# B&R Automation Studio project RS15_RX_30005_r00 (part 7)

#### Control.var
```iecst
(********************************************************************
 * COPYRIGHT -- .
 ********************************************************************
 * Program: Control
 * File: Control.var
 * Author: dominique
 * Created: August 16, 2011
 ********************************************************************
 * Local variables of program Control
 ********************************************************************)

VAR
  bHMI_Bund_ManOn_PB : BOOL ; (*Bundler lacal manuel mode, =0:Off; =1:On*)
  bHMI_Bund_Init_PB  : BOOL ;
  bBundManOn         : BOOL ;
  bBundManOff        : BOOL ;
  bInitBund          : BOOL ;
  bInitBundStart     : BOOL ;
  bInitBundStop      : BOOL ;
  uiBundManTxt_Ind   : UINT ;
  uiBundManCol_Ind   : UINT ;
  uiBundInitTxt_Ind  : UINT ;
  uiBundInitCol_Ind  : UINT ;
  tBundInitTpHorn    : TIME ;

  bHMI_Bund_OnOff  : BOOL ;
  iHMI_BundManLock : INT ;

  H_FB_ToggleTB_0 : H_FB_ToggleTB;

  bBundInit_Perm   : BOOL ;
  H_FB_2StepMove_0 : H_FB_2StepMove ;

  stTP_0 : TP ;
END_VAR

VAR CONSTANT

END_VAR
```

#### ControlInit.st
```iecst
(********************************************************************
 * COPYRIGHT -- .
 ********************************************************************
 * Program: Control
 * File: ControlInit.st
 * Author: dominique
 * Created: August 16, 2011
 ********************************************************************
 * Implementation of program Control
 ********************************************************************)

PROGRAM _INIT

// Bundler Manual/Auto TB Colors
  H_FB_ToggleTB_0.IN_uiTxt0_Ind := 0 ;
  H_FB_ToggleTB_0.IN_uiTxt1_Ind := -1 ;
  H_FB_ToggleTB_0.IN_uiBackCol_State0 := gYellow;
  H_FB_ToggleTB_0.IN_uiForeCol_State0 := gBlack;
  H_FB_ToggleTB_0.IN_uiBackCol_State1 := gGreen;
  H_FB_ToggleTB_0.IN_uiForeCol_State1 := gBlack;

  tBundInitTpHorn     := T#1s ;
  g_tBund_TpWatchSens := T#3s ;

  bHMI_Bund_OnOff := 0 ;

END_PROGRAM
```

### Program Logical/BagMachine_Section/BagBundler/Separator (IEC)

#### SeparatorCyclic.st - Cyclic code
```iecst
(********************************************************************
 * COPYRIGHT -- .
 ********************************************************************
 * Program: Separator
 * File: SeparatorCyclic.st
 * Author: dominique
 * Created: August 15, 2011
 ********************************************************************
 * Implementation of program Separator
 ********************************************************************)

PROGRAM _CYCLIC

    //---------------------------------------------------------------------------------------------------------------------
    // Output assignments
    gQ_Bund_SOL_14C1Out    := bQ_Bund_SOL_14C1Out AND gBagMachine_EstopAlarmsOK ;
    gQ_Bund_SOL_14C2Out    := bQ_Bund_SOL_14C2Out AND gBagMachine_EstopAlarmsOK ;
    gQ_Bund_SOL_PresSelect := bQ_Bund_SOL_PresSelect AND gBagMachine_EstopAlarmsOK ;

    //---------------------------------------------------------------------------------------------------------------------
    // Sensor watching

    H_FB_Flash_0(IN_bEnable:=1, IN_rNumFlashPerSec:=2) ;
    bFlash := H_FB_Flash_0.OUT_bFlash ;

    // S102 on 14C1 Out
    H_FB_WS_14C1.IN_bSensorOut  := gI_Bund_S102 ;
    H_FB_WS_14C1.IN_bSOL_In     := NOT(gQ_Bund_SOL_14C1Out) ;
    H_FB_WS_14C1.IN_bSOL_Out    := gQ_Bund_SOL_14C1Out ;
    H_FB_WS_14C1.IN_bActSensIn  := 0 ;
    H_FB_WS_14C1.IN_bActSensOut := 1 ;
    H_FB_WS_14C1.IN_tTpWatchIn  := g_tBund_TpWatchSens ;
    H_FB_WS_14C1.IN_tTpWatchOut := g_tBund_TpWatchSens ;
    H_FB_WS_14C1.IN_bReset      := gAlarmReset ;
    H_FB_WS_14C1();
    bS102_FaultOut := H_FB_WS_14C1.OUT_bSensOut_FaultOut ;
    bS102_FaultIn  := H_FB_WS_14C1.OUT_bSensOut_FaultIn ;
    bS102_Fault    := H_FB_WS_14C1.OUT_bSensOut_Fault ;

    // S101 on 14C2 In
    H_FB_WS_14C2.IN_bSensorIn   := gI_Bund_S101 ;
    H_FB_WS_14C2.IN_bSOL_In     := NOT(gQ_Bund_SOL_14C2Out) ;
    H_FB_WS_14C2.IN_bSOL_Out    := gQ_Bund_SOL_14C2Out ;
    H_FB_WS_14C2.IN_bActSensIn  := 1 ;
    H_FB_WS_14C2.IN_bActSensOut := 0 ;
    H_FB_WS_14C2.IN_tTpWatchIn  := g_tBund_TpWatchSens ;
    H_FB_WS_14C2.IN_tTpWatchOut := g_tBund_TpWatchSens ;
    H_FB_WS_14C2.IN_bReset      := gAlarmReset ;
    H_FB_WS_14C2();
    bS101_FaultOut := H_FB_WS_14C2.OUT_bSensIn_FaultOut ;
    bS101_FaultIn  := H_FB_WS_14C2.OUT_bSensIn_FaultIn ;
    bS101_Fault    := H_FB_WS_14C2.OUT_bSensIn_Fault ;

    // HMI Sensors states display
    IF gI_Bund_S101 THEN
      iHMI_Bund_S101 := 1 ;
    ELSE
      iHMI_Bund_S101 := 0 ;
    END_IF
    IF bS101_Fault AND
       bFlash      THEN
      iHMI_Bund_S101 := 2 ;
    END_IF

    IF gI_Bund_S102 THEN
      iHMI_Bund_S102 := 1 ;
    ELSE
      iHMI_Bund_S102 := 0 ;
    END_IF
    IF bS102_Fault AND
       bFlash      THEN
      iHMI_Bund_S102 := 2 ;
    END_IF

    IF gI_Bund_S103 THEN
      iHMI_Bund_S103 := 1 ;
    ELSE
      iHMI_Bund_S103 := 0 ;
    END_IF

    IF gI_Bund_S109 THEN
      iHMI_Bund_S109 := 1 ;
    ELSE
      iHMI_Bund_S109 := 0 ;
    END_IF

    g_bBund_SensFaultCycSep := bS101_Fault OR bS102_Fault ;

    // HMI Cylinders states display
    // Cylinder 14C1
    // Case Out
    IF gQ_Bund_SOL_14C1Out THEN
      iHMI_Bund_14C1Out_State := 4 ;
      iHMI_Bund_14C1In_State  := 0 ;
    END_IF
    IF bS102_FaultOut THEN
      IF bFlash THEN
        iHMI_Bund_14C1Out_State := 5 ;
      ELSE
        iHMI_Bund_14C1Out_State := 6 ;
      END_IF
    END_IF
    // Case In
    IF NOT(gQ_Bund_SOL_14C1Out) THEN
      iHMI_Bund_14C1In_State  := 1 ;
      iHMI_Bund_14C1Out_State := 0 ;
    END_IF
    IF bS102_FaultIn THEN
      IF bFlash THEN
        iHMI_Bund_14C1In_State := 2 ;
      ELSE
        iHMI_Bund_14C1In_State := 3 ;
      END_IF
    END_IF

    // Cylinder 14C2
    // Case Out
    IF gQ_Bund_SOL_14C2Out THEN
      iHMI_Bund_14C2Out_State := 4 ;
      iHMI_Bund_14C2In_State  := 0 ;
    END_IF
    IF bS101_FaultOut THEN
      IF bFlash THEN
        iHMI_Bund_14C2Out_State := 5 ;
      ELSE
        iHMI_Bund_14C2Out_State := 6 ;
      END_IF
    END_IF
    // Case In
    IF NOT(gQ_Bund_SOL_14C2Out) THEN
      iHMI_Bund_14C2In_State  := 1 ;
      iHMI_Bund_14C2Out_State := 0 ;
    END_IF
    IF bS101_FaultIn THEN
      IF bFlash THEN
        iHMI_Bund_14C2In_State := 2 ;
      ELSE
        iHMI_Bund_14C2In_State := 3 ;
      END_IF
    END_IF

    // Pressure selection PB
    IF bQ_Bund_SOL_PresSelect THEN
      uiPresSelPBTxt_Id := 1 ;
      uiPresSelPBCol_Id := 197 + gBlack * 256 ;
    ELSE
      uiPresSelPBTxt_Id := 0 ;
      uiPresSelPBCol_Id := 42 + gBlack * 256 ;
    END_IF ;

    //---------------------------------------------------------------------------------------------------------------------
    // Packet separator cycle
    //---------------------------------------------------------------------------------------------------------------------

    // Start cycle
    IF g_bIndSelBundProd              AND
       gBagMachine_EstopAlarmsOK      AND
       NOT(bInitSepCycl)              AND
       NOT(g_bBund_SensFaultCycSep)   AND
       NOT(g_bBund_TimOutFaultCycSep) AND
       1                              THEN
      stCycBundSep.bSCyc := 1 ;
    END_IF ;

    //----------------------------------------------------------------------
    // Cycle at rest
    IF NOT(stCycBundSep.bSCyc) AND
       1                       THEN
      IF NOT( stCycBundSep.bFCyc ) THEN
        // Init after cycle unpropaly ended
        stCycBundSep.bFCyc := 1 ;
        stCycBundSep.bCyc  := 0 ;
        stCycBundSep.bCycFail := 1 ;

        bInitSepCycl    := 0 ;
        g_bBund_InitSep := 0 ;
      END_IF
      stCycBundSep.iStep := 0 ;
      RETURN ;
    ELSE
    //----------------------------------------------------------------------
    // Cycle running

    // Manu mode
      IF g_bIndBundManu THEN
        stCycBundSep.iStep := C_iSTEP_15 ;
        // In manu mode cycle is frozen in Step15
        IF bHMI_BundMan_14C1P_PB THEN
          bQ_Bund_SOL_14C1Out := 1 ;
        END_IF
        IF bHMI_BundMan_14C1M_PB THEN
          bQ_Bund_SOL_14C1Out := 0 ;
        END_IF
        IF bHMI_BundMan_14C2P_PB THEN
          bQ_Bund_SOL_14C2Out := 1 ;
        END_IF
        IF bHMI_BundMan_14C2M_PB THEN
          bQ_Bund_SOL_14C2Out := 0 ;
        END_IF
        IF bHMI_BundMan_PresSelect_PB THEN
          bQ_Bund_SOL_PresSelect := NOT(bQ_Bund_SOL_PresSelect) ;
          bHMI_BundMan_PresSelect_PB := 0 ;
          iTest := iTest + 1 ;
        END_IF
      END_IF
      IF NOT(g_bIndBundManu) THEN
        bHMI_BundMan_14C1P_PB := 0 ;
        bHMI_BundMan_14C2P_PB := 0 ;
        bHMI_BundMan_14C1M_PB := 0 ;
        bHMI_BundMan_14C2M_PB := 0 ;
        bHMI_BundMan_PresSelect_PB := 0 ;
      END_IF

    // Permanent conditions
      IF NOT(gBagMachine_EstopAlarmsOK) OR
         g_bBund_SensFaultCycSep        THEN
        stCycBundSep.bSCyc := 0 ;
        bHMI_BundMan_14C1P_PB := 0 ;
        bHMI_BundMan_14C2P_PB := 0 ;
        bHMI_BundMan_14C1M_PB := 0 ;
        bHMI_BundMan_14C2M_PB := 0 ;
        bHMI_BundMan_PresSelect_PB := 0 ;
      END_IF

      // Init cycle
      // Start init
      IF g_bBund_InitSep   AND
         NOT(bInitSepCycl) THEN
        bInitSepCycl      := 1 ;
        g_bBundInitSep_OK := 0 ;
        g_bBund_ResetCountReq := 1 ;
        // Put cycle in Step 4
        stCycBundSep.iStep := C_iSTEP_4 ;
        // Action Step 4
        bQ_Bund_SOL_14C1Out := 0 ;

        // Init cycle
        stCycBundSep.bFCyc := 0 ;
        stCycBundSep.bCyc  := 1 ;
        stCycBundSep.bCycFail := 0 ;
        iMemoStepCyc := C_iSTEP_99 ;
      END_IF
      // Stop init
      IF g_bBundStopInitSep THEN
        g_bBund_InitSep    := 0 ;
        g_bBundInitSep_OK  := 0 ;
        g_bBundStopInitSep := 0 ;
        stCycBundSep.bSCyc := 0 ;
      END_IF

      // Watching Step time out
      IF g_bIndBundManu                     OR
         ( stCycBundSep.iStep < C_iSTEP_4 ) THEN
        iMemoStepCyc := C_iSTEP_99 ;
        stTON_WatchCyc(IN:=(iMemoStepCyc=stCycBundSep.iStep), PT:=tTpWatchCyc);
      ELSE
        stTON_WatchCyc(IN:=(iMemoStepCyc=stCycBundSep.iStep), PT:=tTpWatchCyc);
        iMemoStepCyc := stCycBundSep.iStep ;
      END_IF
      IF stTON_WatchCyc.Q THEN
        g_bBund_TimOutFaultCycSep := 1 ;
        stCycBundSep.bSCyc := 0 ;
      END_IF

    // Permanent actions
      stTON_RetCyl14C1(IN:=(stCycBundSep.iStep = C_iSTEP_4), PT:=tTpRetCyl14C1) ;

      // Selection pressure in contre-weight cylinder of Separator
      // bQ_Bund_SOL_PresSelect = 1 => pressure contre-weight
      // bQ_Bund_SOL_PresSelect = 0 => supply pressure
      stTON_SelPres(IN:=bQ_Bund_SOL_14C2Out, PT:=tTpSelPres) ;
      IF NOT(g_bIndBundManu) THEN
        bQ_Bund_SOL_PresSelect := stTON_SelPres.Q ;
      END_IF
    END_IF
    //----------------------------------------------------------------------
    // Cycle steps

        CASE stCycBundSep.iStep OF

        C_iSTEP_0 :
         //----------------------------------------------
         // Etape 1 : Initialisation cycle
         //----------------------------------------------
          IF TRUE THEN
            stCycBundSep.iStep := C_iSTEP_1 ;

            // Action Step 1
            stCycBundSep.bFCyc := 0 ;
            stCycBundSep.bCyc  := 1 ;
            stCycBundSep.bCycFail := 0 ;

            bQ_Bund_SOL_14C1Out := 1 ;
            bQ_Bund_SOL_14C2Out := 0 ;
            g_bBundPackCountOK  := 0 ;
          END_IF

        C_iSTEP_1 :
         //----------------------------------------------
         // Etape 2 : Waiting for pack count
         //----------------------------------------------
          IF gI_Bund_S101                   AND
             gI_Bund_S102                   AND
             ( stCycBundSep.bTestOn         OR
               NOT(stCycBundSep.bModTest) ) THEN
            stCycBundSep.iStep := C_iSTEP_2 ;

            // Action Step 2
            stCycBundSep.bTestOn := 0 ;

            // Waiting for pack count
          END_IF

        C_iSTEP_2 :
         //----------------------------------------------
         // Step 3 : Out cylinder 14C2 to separate packet
         //          and activate tempo in permanent actions for contre-weight pressure selection
         //          and waiting for sensor S103
         //----------------------------------------------
          IF g_bBundPackCountOK             AND
             g_bBundInitSep_OK              AND
             ( stCycBundSep.bTestOn         OR
               NOT(stCycBundSep.bModTest) ) THEN
            stCycBundSep.iStep := C_iSTEP_3 ;

            // Action Step 3
            stCycBundSep.bTestOn := 0 ;

            bQ_Bund_SOL_14C2Out := 1 ;
            g_bBundPackCountOK  := 0 ;
          END_IF

        C_iSTEP_3 :
         //----------------------------------------------
         // Step 4 : Move in cylinder 14C1
         //          and activate tempo in permanent actions
         //----------------------------------------------
          IF g_bBund_MoveInSep_OK           AND
             ( stCycBundSep.bTestOn         OR
               NOT(stCycBundSep.bModTest) ) THEN
            stCycBundSep.iStep := C_iSTEP_4 ;

            // Action Step 4
            stCycBundSep.bTestOn := 0 ;

            bQ_Bund_SOL_14C1Out  := 0 ;
            g_bBund_MoveInSep_OK := 0 ;
          END_IF

        C_iSTEP_4 :
         //----------------------------------------------
         // Step 5 : Move in cylinder 14C2 to put back separator in init position
         //----------------------------------------------
          IF stTON_RetCyl14C1.Q             AND
             ( stCycBundSep.bTestOn         OR
               NOT(stCycBundSep.bModTest) ) THEN
            stCycBundSep.iStep := C_iSTEP_5 ;

            // Action Step 5
            stCycBundSep.bTestOn := 0 ;

            bQ_Bund_SOL_14C2Out := 0 ;
          END_IF

        C_iSTEP_5 :
         //----------------------------------------------
         // Step 6 : Output cylinder 14C1 to out the separation fingers
         //----------------------------------------------
          IF gI_Bund_S101                   AND
             ( stCycBundSep.bTestOn         OR
               NOT(stCycBundSep.bModTest) ) THEN
            stCycBundSep.iStep := C_iSTEP_6 ;

            // Action Step 6
            stCycBundSep.bTestOn := 0 ;

            bQ_Bund_SOL_14C1Out := 1 ;
          END_IF

        C_iSTEP_6 :
         //----------------------------------------------
         // Etape 2 : Waiting for pack count
         //----------------------------------------------
          IF gI_Bund_S102                   AND
             ( stCycBundSep.bTestOn         OR
               NOT(stCycBundSep.bModTest) ) THEN
            stCycBundSep.iStep := C_iSTEP_2 ;

            // Action Step 2
            stCycBundSep.bTestOn := 0 ;
            // Waiting for pack count

            g_bBund_InitSep   := 0 ;
            bInitSepCycl      := 0 ;
            g_bBundInitSep_OK := 1 ;
          END_IF

        C_iSTEP_15 :
         //----------------------------------------------
         // Etape 1 : Initialisation cycle
         //----------------------------------------------
          IF NOT(g_bIndBundManu)            AND
             ( stCycBundSep.bTestOn         OR
               NOT(stCycBundSep.bModTest) ) THEN
            stCycBundSep.iStep := C_iSTEP_1 ;

            // Action Step 1
            stCycBundSep.bTestOn := 0 ;

            stCycBundSep.bFCyc := 0 ;
            stCycBundSep.bCyc  := 1 ;

            g_bBundPackCountOK  := 0 ;
            // Waiting for pack count
          END_IF
        END_CASE
    //---------------------------------------------------------------------------------------------------------------------

END_PROGRAM
```

#### SeparatorInit.st - Initialization code
```iecst
(********************************************************************
 * COPYRIGHT -- .
 ********************************************************************
 * Program: Separator
 * File: SeparatorInit.st
 * Author: dominique
 * Created: August 15, 2011
 ********************************************************************
 * Implementation of program Separator
 ********************************************************************)

PROGRAM _INIT

(* TODO : Add your code here *)
  tTpRetCyl14C1         := T#1s ;
  tTpWatchCyc           := T#6s ;
  tTpSelPres            := T#0.5s ;
  stCycBundSep.bModTest := 0 ;
  stCycBundSep.bTestOn  := 0 ;

END_PROGRAM
```

- Program Logical/BagMachine_Section/BagBundler/Test_Simul (IEC) (no source held here)

### Program Logical/BagMachine_Section/BagBundler/Tilter (IEC)

#### TilterInit.st - Initialization code
```iecst
(********************************************************************
 * COPYRIGHT -- .
 ********************************************************************
 * Program: Tilting
 * File: TiltingInit.st
 * Author: dominique
 * Created: August 16, 2011
 ********************************************************************
 * Implementation of program Tilting
 ********************************************************************)

PROGRAM _INIT

(* TODO : Add your code here *)
  rPosTiltDegPts := gr_rPosTiltTravel/C_rMaxAna ;
  rK := 1 ;
  rK_HMI := 35 ;
  rPosTiltInit_OK  := 1.0 ;
  rPosTiltInitHyst := 0.5 ;
  tTpStopTilt      := T#0.5s ;
  tTpOut14C5       := T#0.5s ;
  tTpOut14C3       := T#1s ;
  tTpWatchCyc      := T#6s ;

END_PROGRAM
```

### Program Logical/BagMachine_Section/Count (IEC) - Accurate Product Count Code

#### Count.var
```iecst
(********************************************************************
 * COPYRIGHT --
 ********************************************************************
 * Program: Count
 * File: Count.var
 * Author: pkiel
 * Created: October 21, 2009
 ********************************************************************
 * Local variables of program Count
 ********************************************************************)
VAR
	Count_On : BOOL;
	Count_PB : BOOL;
	CountPBColor_Ind : UINT;
	CountPBText_Ind : UINT;
	CountPulse : BOOL;
	CurrentPackCount : DINT;
  iCurrentpackCountTilt : INT;
  iBagCountStartTilt : INT;
  stTON_S103_Filtr   : TON ;
  tTpS103Filtr       : TIME ;
END_VAR
VAR RETAIN
	HGW_2StatePB_0 : HGW_2StatePB;
END_VAR
VAR
	HMI_CountSelect_Ind : UINT;
	HMI_CountSelect_PB : BOOL;
	HMI_ProductCount : DINT;
	HMI_ProductCountReset_PB : BOOL;
	HMI_ProductCountVisibility : UINT;
END_VAR
VAR RETAIN
	PackCount : DINT;
	ProductCount1 : DINT;
	ProductCount2 : DINT;
	ProductCount3 : DINT;
	ProductCount4 : DINT;
END_VAR
VAR
	TriggerCount : DINT;
END_VAR
```

#### CountCyclic.st
```iecst
(********************************************************************
 * COPYRIGHT --
 ********************************************************************
 * Program: Count
 * File: CountCyclic.st
 * Author: pkiel
 * Created: October 21, 2009
 ********************************************************************
 * Implementation of program Count
 ********************************************************************)

PROGRAM _CYCLIC

(* Hand Count Setpoints & Limits *)
	gRecipeActive.PackCount:=LIMIT(0,gRecipeActive.PackCount,32767);
	gRecipeActive.HoldCount:=LIMIT(0,gRecipeActive.HoldCount,gRecipeActive.PackCount);
	TriggerCount:=gRecipeActive.PackCount-gRecipeActive.HoldCount;

(* Generate Count Pulse From Master Axis *)
	IF (gA[9].PositionDeg>0 AND gA[9].PositionDeg<90) THEN
		CountPulse := 1;
	END_IF
	IF (gA[9].PositionDeg>180 AND gA[9].PositionDeg<240) THEN
		CountPulse := 0;
	END_IF

(* Product Count *)
	IF(EDGEPOS(CountPulse)) THEN
		CurrentPackCount:=CurrentPackCount+1;
    iCurrentpackCountTilt := iCurrentpackCountTilt + 1 ;   //modif increment compt sac apres s103
    // Master number of revolutions
    gA[9].uiiNumRev := gA[9].uiiNumRev + 1 ;
    IF gA[9].uiiNumRev < 0 THEN
      gA[9].uiiNumRev := 0 ;
    END_IF
		IF (gSP_TubeSelect) THEN
			ProductCount1:=ProductCount1+2;
			ProductCount2:=ProductCount2+2;
			ProductCount3:=ProductCount3+2;
			ProductCount4:=ProductCount4+2;
		ELSE
			ProductCount1:=ProductCount1+1;
			ProductCount2:=ProductCount2+1;
			ProductCount3:=ProductCount3+1;
			ProductCount4:=ProductCount4+1;
		END_IF
	END_IF

(* Count Off/On From HMI *)
	HGW_2StatePB_0.PB := EDGEPOS(Count_PB);
	CountPBText_Ind := HGW_2StatePB_0.Text_Ind;
	CountPBColor_Ind := HGW_2StatePB_0.Color_Ind;
	Count_On := HGW_2StatePB_0.State1;
	HGW_2StatePB_0();

(* Delivery Bag Count Solenoid...Disable Count SOL If HandCount Setpoint = 0*)
	IF (gRecipeActive.PackCount>0 AND Count_On) THEN
		IF (CurrentPackCount>=TriggerCount) THEN
			gQ_SOL_BagCount:=1;
		ELSE
			gQ_SOL_BagCount:=0;
		END_IF
	ELSE
		gQ_SOL_BagCount:=0;
	END_IF

(* Pack Count Evaluation *)
  IF (CurrentPackCount>=gRecipeActive.PackCount) THEN
    CurrentPackCount := 0 ;
    g_bBundPackCountOK := (gRecipeActive.PackCount > 0) ;
		IF (gSP_TubeSelect) THEN
			PackCount:=PackCount+2;
		ELSE
			PackCount:=PackCount+1;
		END_IF
  END_IF
  // Bundler reset bag count requested
  IF g_bBund_ResetCountReq THEN
    CurrentPackCount := 0 ;
    g_bBund_ResetCountReq := 0 ;
  END_IF

  //*****************************************D.M. 29092011  BrownPaper_14543  change proram
(*start tilter with counter*)
         iBagCountStartTilt := LIMIT(0,gHMI_Bund_iBagCountStartTilt,40);

         stTON_S103_Filtr(IN:=gI_Bund_S103, PT:=tTpS103Filtr) ;
         IF NOT(gI_Bund_S103) THEN
           iCurrentpackCountTilt := 0;
           g_bBund_StartTilt := 0 ;
         END_IF

         IF EDGEPOS(iCurrentpackCountTilt>=iBagCountStartTilt)       OR
            EDGEPOS(stTON_S103_Filtr.Q) AND (iBagCountStartTilt = 0) THEN
           g_bBund_StartTilt := 1;
         END_IF

   //*****************************************End D.M. 29092011  BrownPaper_14543  change proram

(* Product Count Limits *)
	IF (ProductCount1>=2147483646) THEN
		ProductCount1:=0;
	END_IF
	IF (ProductCount2>=2147483646) THEN
		ProductCount2:=0;
	END_IF
	IF (ProductCount3>=2147483646) THEN
		ProductCount3:=0;
	END_IF
	IF (ProductCount4>=2147483646) THEN
		ProductCount4:=0;
	END_IF

(* HMI Count Display *)

	IF (HMI_CountSelect_PB) THEN
		HMI_CountSelect_Ind:=HMI_CountSelect_Ind+1;
		IF (HMI_CountSelect_Ind>5) THEN
			HMI_CountSelect_Ind:=1;
		END_IF
		HMI_CountSelect_PB:=0;
	END_IF

	CASE (HMI_CountSelect_Ind) OF
		1:
			HMI_ProductCount:=ProductCount1;
			IF (HMI_ProductCountReset_PB) THEN
				ProductCount1:=0;
				HMI_ProductCountReset_PB:=0;
			END_IF
		2:
			HMI_ProductCount:=ProductCount2;
			IF (HMI_ProductCountReset_PB) THEN
				ProductCount2:=0;
				HMI_ProductCountReset_PB:=0;
			END_IF
		3:
				HMI_ProductCount:=ProductCount3;
			IF (HMI_ProductCountReset_PB) THEN
				ProductCount3:=0;
				HMI_ProductCountReset_PB:=0;
			END_IF
		4:
			HMI_ProductCount:=ProductCount4;
			IF (HMI_ProductCountReset_PB) THEN
				ProductCount4:=0;
				HMI_ProductCountReset_PB:=0;
			END_IF
		5:
			HMI_ProductCount:=PackCount;
			IF (HMI_ProductCountReset_PB) THEN
				PackCount:=0;
				HMI_ProductCountReset_PB:=0;
			END_IF
	END_CASE

END_PROGRAM
```

#### CountInit.st
```iecst
(********************************************************************
 * COPYRIGHT --
 ********************************************************************
 * Program: Count
 * File: CountInit.st
 * Author: pkiel
 * Created: October 21, 2009
 ********************************************************************
 * Implementation of program Count
 ********************************************************************)

PROGRAM _INIT

	HMI_CountSelect_Ind:=LIMIT(1,HMI_CountSelect_Ind,5);
	HMI_ProductCountVisibility:=1;

(* Count Off/On PB Colors *)
	HGW_2StatePB_0.BackColor_State0 := gBlue;
	HGW_2StatePB_0.ForeColor_State0 := gWhite;
	HGW_2StatePB_0.BackColor_State1 := gGreen;
	HGW_2StatePB_0.ForeColor_State1 := gBlack;

END_PROGRAM
```

### Program Logical/BagMachine_Section/HotGlue (IEC) - Hot Glue Seam Paste Control

#### HotGlue.var
```iecst
(********************************************************************
 * COPYRIGHT -- Microsoft
 ********************************************************************
 * Program: HotGlue
 * File: HotGlue.var
 * Author: pkiel
 * Created: July 14, 2011
 ********************************************************************
 * Local variables of program HotGlue
 ********************************************************************)
VAR
	Glue_Auto : BOOL;
	Glue_On : BOOL;
	Glue_PB : BOOL;
	GlueAuto_On : BOOL;
	GlueAuto_PB : BOOL;
	GlueAutoColor_Ind : UINT;
	GlueAutoText_Ind : UINT;
	GlueClean_PB : BOOL;
	GlueColor_Ind : UINT;
	GluePurge_PB : BOOL;
	GlueText_Ind : UINT;
END_VAR
VAR RETAIN
	HGW_2StatePB_0 : HGW_2StatePB;
	HGW_2StatePB_1 : HGW_2StatePB;
  HMI_bSelHotColdRSGlue_PB : BOOL ;
END_VAR
VAR
	HGW_ScaleReal_0 : HGW_ScaleReal;
	HGW_ScaleReal_1 : HGW_ScaleReal;
	HGW_Toggle_0 : HGW_Toggle;
	PressureCmd : REAL;
END_VAR
```

#### HotGlueInit.st
```iecst
(********************************************************************
 * COPYRIGHT -- Microsoft
 ********************************************************************
 * Program: HotGlue
 * File: HotGlueInit.st
 * Author: pkiel
 * Created: July 14, 2011
 ********************************************************************
 * Implementation of program HotGlue
 ********************************************************************)

PROGRAM _INIT

(* Glue Off/On PB Colors *)
	HGW_2StatePB_0.BackColor_State0 := gBlue;
	HGW_2StatePB_0.ForeColor_State0 := gWhite;
	HGW_2StatePB_0.BackColor_State1 := gGreen;
	HGW_2StatePB_0.ForeColor_State1 := gBlack;

(* Glue Manual/Auto PB Colors *)
	HGW_2StatePB_1.BackColor_State0 := gYellow;
	HGW_2StatePB_1.ForeColor_State0 := gBlack;
	HGW_2StatePB_1.BackColor_State1 := gGreen;
	HGW_2StatePB_1.ForeColor_State1 := gBlack;

END_PROGRAM
```

### Program Logical/BagMachine_Section/RS_Glue (IEC) - Cold Glue Seam Paste Control

#### RS_Glue.var - Local variables
```iecst
(********************************************************************
 * COPYRIGHT -- Microsoft
 ********************************************************************
 * Program: RS_Glue
 * File: RS_Glue.var
 * Author: dominique
 * Created: October 26, 2011
 ********************************************************************
 * Local variables of program ColdGlue
 ********************************************************************)
VAR
	Glue_Auto         : BOOL;
	Glue_On           : BOOL;
	Glue_PB           : BOOL;
	GlueAuto_On       : BOOL;
	GlueAuto_PB       : BOOL;
	GlueAutoColor_Ind : UINT;
	GlueAutoText_Ind  : UINT;
	GlueColor_Ind     : UINT;
	GluePurge_PB      : BOOL;
	GlueText_Ind      : UINT;
  rGlueMinPress     : REAL ;
  rGlueMaxPress     : REAL ;
  bTest1            : BOOL ;
  bTest2            : BOOL ;

END_VAR
VAR RETAIN
	HGW_2StatePB_0 : HGW_2StatePB;
	HGW_2StatePB_1 : HGW_2StatePB;
  stSP_ColdGlue : Glue ;
  stSP_HotGlue  : Glue ;
END_VAR
VAR
	HGW_ScaleReal_0 : HGW_ScaleReal;
	HGW_ScaleReal_1 : HGW_ScaleReal;
	PressureCmd : REAL;
	GlueClean_PB : BOOL;
	HGW_Toggle_0 : HGW_Toggle;
END_VAR
```

- Program Logical/BagMachine_Section/RS_Glue_V0 (IEC) - Cold Glue Seam Paste Control (no source held here)

### Program Logical/BagMachine_Section/Unw_3W_Glue (IEC) - Hot Glue Seam Paste Control

#### Unw_3W_GlueCyclic.st
```iecst
(********************************************************************
 * COPYRIGHT -- Microsoft
 ********************************************************************
 * Program: Unw_3W_Glue
 * File: Unw_3W_Glue.st
 * Author: dominique
 * Created: October 26, 2011
 ********************************************************************
 * Implementation of program Unw_3W_Glue
 ********************************************************************)

PROGRAM _CYCLIC

  // Limit operator setpoint
  gSP_OtherRSGlue.MinPressure := LIMIT (0,gSP_OtherRSGlue.MinPressure,399) ;
  gSP_OtherRSGlue.MaxPressure := LIMIT (0,gSP_OtherRSGlue.MaxPressure,400) ;

  // Type glue selection (Cold/Hot)

  gRecipeActive.bSelTypeOtherRSGlue := 1 ; // D.M. Le 09/12/2011 Pyrollpack_14661 sur DHS uniquement colle chaude, pas de colle froide

  gQ_CR_HotColdOtherRSGlueSelect := gRecipeActive.bSelTypeOtherRSGlue ;
  IF EDGEPOS(gRecipeActive.bSelTypeOtherRSGlue) THEN
    // Switch set points on screen from Cold to Hot
    stSP_ColdGlue.MinPressure := gSP_OtherRSGlue.MinPressure ;
    stSP_ColdGlue.MaxPressure := gSP_OtherRSGlue.MaxPressure ;
    stSP_ColdGlue.ManPressure := gSP_OtherRSGlue.ManPressure ;
    stSP_ColdGlue.AutoOnSpeed := gSP_OtherRSGlue.AutoOnSpeed ;

    gSP_OtherRSGlue.MinPressure := stSP_HotGlue.MinPressure ;
    gSP_OtherRSGlue.MaxPressure := stSP_HotGlue.MaxPressure ;
    gSP_OtherRSGlue.ManPressure := stSP_HotGlue.ManPressure ;
    gSP_OtherRSGlue.AutoOnSpeed := stSP_HotGlue.AutoOnSpeed ;
  END_IF ;
  IF EDGENEG(gRecipeActive.bSelTypeOtherRSGlue) THEN
    // Switch set points on screen from Hot to Cold
    stSP_HotGlue.MinPressure := gSP_OtherRSGlue.MinPressure ;
    stSP_HotGlue.MaxPressure := gSP_OtherRSGlue.MaxPressure ;
    stSP_HotGlue.ManPressure := gSP_OtherRSGlue.ManPressure ;
    stSP_HotGlue.AutoOnSpeed := gSP_OtherRSGlue.AutoOnSpeed ;

    gSP_OtherRSGlue.MinPressure := stSP_ColdGlue.MinPressure ;
    gSP_OtherRSGlue.MaxPressure := stSP_ColdGlue.MaxPressure ;
    gSP_OtherRSGlue.ManPressure := stSP_ColdGlue.ManPressure ;
    gSP_OtherRSGlue.AutoOnSpeed := stSP_ColdGlue.AutoOnSpeed ;
  END_IF ;

(* Glue Off/On From HMI *)
  HGW_2StatePB_0.PB := EDGEPOS(Glue_PB);
  GlueText_Ind := HGW_2StatePB_0.Text_Ind;
  GlueColor_Ind := HGW_2StatePB_0.Color_Ind;
  Glue_On := HGW_2StatePB_0.State1;
  HGW_2StatePB_0();

(* Glue Manual/Auto From HMI *)
	HGW_2StatePB_1.PB := (EDGEPOS(GlueAuto_PB) OR (NOT Glue_Auto AND gA[9].Ind_InMotion));
	GlueAutoText_Ind := HGW_2StatePB_1.Text_Ind;
	GlueAutoColor_Ind := HGW_2StatePB_1.Color_Ind;
	Glue_Auto := HGW_2StatePB_1.State1;
	HGW_2StatePB_1();

(* Glue Auto Pressure Based On Machine Speed *)
	HGW_ScaleReal_0.Enable := Glue_Auto;
	HGW_ScaleReal_0.InputMin := 0.0;
	HGW_ScaleReal_0.InputMax := gr_rMaxLSFlexoP_mmin/3.2808;
	HGW_ScaleReal_0.InputRaw := gActualMachineSpeed_FPM;
	HGW_ScaleReal_0.ScaledMin := gSP_OtherRSGlue.MinPressure ;
	HGW_ScaleReal_0.ScaledMax := gSP_OtherRSGlue.MaxPressure ;
	PressureCmd := HGW_ScaleReal_0.ScaledOut;
	HGW_ScaleReal_0();

(* Glue Manual Pressure *)
	IF (NOT Glue_Auto) THEN
		PressureCmd := gSP_OtherRSGlue.ManPressure;
	END_IF

(* Glue Pressure Command Limit 0-100% *)
	PressureCmd := LIMIT (0,PressureCmd, 100);

(* If Disabled, Reduce Pressure To Zero *)
	IF (NOT Glue_On) THEN
		PressureCmd := 0;
	END_IF

(* Generate Analog Command To Seam Paste System Pressure *)
	HGW_ScaleReal_1.Enable := 1;
	HGW_ScaleReal_1.InputMin := 0.0;
	HGW_ScaleReal_1.InputMax := 100.0;
	HGW_ScaleReal_1.InputRaw := PressureCmd;
	HGW_ScaleReal_1.ScaledMin := 0.0;
	HGW_ScaleReal_1.ScaledMax := 32767.0;
  HMI_rOtherRSGlueActPress := REAL_TO_INT(HGW_ScaleReal_1.ScaledOut)/32767.0*100.0;

  gQ_CMD_UNW_GluePressure := REAL_TO_INT(HGW_ScaleReal_1.ScaledOut);
  gQ_CMD_3W_GluePressure  := REAL_TO_INT(HGW_ScaleReal_1.ScaledOut);
  gQ_CMD_OtherRS_GluePressure := REAL_TO_INT(HGW_ScaleReal_1.ScaledOut);
	HGW_ScaleReal_1();

  // Delay activation glue
    // Limit operator value
    HMI_rSPDelayActGlue := LIMIT(0,HMI_rSPDelayActGlue,10) ;
    // Conversion from s --> ms in time format
    iiSPDelayActGlue := REAL_TO_DINT(HMI_rSPDelayActGlue*1000) ;
    tSPDelayActGlue := DINT_TO_TIME(iiSPDelayActGlue) ;
    // Delay calculation
    stTON_DelayActGlue(IN:=(gA[9].Ind_InMotion AND gA[5].Ind_bSynchroOK), PT:=tSPDelayActGlue);

    // Glue activation/deactivation
    GlueAuto_On := gI_SS_UNW_HotGlue    AND
                   stTON_DelayActGlue.Q ;

  (* Glue Gun Clean Control *)
  	HGW_Toggle_0(In := GlueClean_PB , Time := T#12ms);

  (* Glue Gun Control *)
  	IF (GlueAuto_On OR GluePurge_PB OR HGW_Toggle_0.Out) THEN
  		bImQ_CR_UNW_Glue := 1;
  	ELSE
  		bImQ_CR_UNW_Glue := 0;
  	END_IF

    // Output activation
    // Glue on unwinder
    gQ_CR_UNW_Glue := bImQ_CR_UNW_Glue AND
                      NOT(g_bIndEStop) ;

    // Glue on 3Web unit
    Glue3WAuto_On := stTON_DelayActGlue.Q   AND
                     gBagMachine_WebBreakOK AND
                     g_bSynchroAxisOK       ;

    bQ_CR_3W_GlueOn := ( Glue3WAuto_On      OR
                         GluePurge_PB       OR
                         HGW_Toggle_0.Out ) AND
                       gI_SS_3W_GlueOn      ;

    bQ_CR_3W_Glue2 := gI_SS_3W_Glue2  AND
                      bQ_CR_3W_GlueOn ;

    // Outputs activation
    gQ_CR_3W_GlueOn := bQ_CR_3W_GlueOn AND
                       NOT(g_bIndEStop) ;
    gQ_CR_3W_Glue2 := bQ_CR_3W_Glue2 AND
                      NOT(g_bIndEStop) ;
END_PROGRAM
```

### Program Logical/BagMachine_Section/GlueTray (IEC) - Glue Tray Control

#### GlueTrayCyclic.st - Cyclic code
```iecst
(********************************************************************
 * COPYRIGHT -- Microsoft
 ********************************************************************
 * Program: GlueTray
 * File: GlueTrayCyclic.st
 * Author: pkiel
 * Created: July 19, 2011
 ********************************************************************
 * Implementation of program GlueTray
 ********************************************************************)

PROGRAM _CYCLIC

(* Glue Tray Man/Auto From HMI *)
	HGW_2StatePB_0.PB := EDGEPOS(GlueTray_PB);
	GlueTrayText_Ind := HGW_2StatePB_0.Text_Ind;
	GlueTrayColor_Ind := HGW_2StatePB_0.Color_Ind;
	GlueTray_Auto := HGW_2StatePB_0.State1;
	HGW_2StatePB_0();

(* Limit Glue Tray Auto On Speed *)
	gSP_GlueTrayAutoSpeed := LIMIT(12,gSP_GlueTrayAutoSpeed,500);

(* Glue Tray Man/Auto Control *)
	CASE (GlueTrayText_Ind) OF
		0: (* Manual Control *)
			IF (gI_SS_GluePanUpDown) THEN
				gQ_SOL_GluePan := 1;
			ELSE
				gQ_SOL_GluePan := 0;
			END_IF

		1: (* Auto Control *)
			IF (gI_SS_GluePanUpDown AND
				gActualMachineSpeed_FPM>gSP_GlueTrayAutoSpeed) THEN
				gQ_SOL_GluePan := 1;
			ELSE
				gQ_SOL_GluePan := 0;
			END_IF
	END_CASE

(* Glue Tray Slow Rotation On/Off From HMI *)
	HGW_2StatePB_1.PB := EDGEPOS(GlueTraySR_PB);
	GlueTraySRText_Ind := HGW_2StatePB_1.Text_Ind;
	GlueTraySRColor_Ind := HGW_2StatePB_1.Color_Ind;
	GlueTraySR_On := HGW_2StatePB_1.State1;
	HGW_2StatePB_1();

(* Glue Tray Slow Rotation Control *)
	IF (GlueTraySR_On AND gI_SafetyRelay_EStopOK AND gQ_CR_MainPowerOn) THEN
		gQ_CON_GlueSlowRotation := 1;
	ELSE
		gQ_CON_GlueSlowRotation := 0;
	END_IF

END_PROGRAM
```

#### GlueTrayInit.st - Initialization code
```iecst
(********************************************************************
 * COPYRIGHT -- Microsoft
 ********************************************************************
 * Program: GlueTray
 * File: GlueTrayInit.st
 * Author: pkiel
 * Created: July 19, 2011
 ********************************************************************
 * Implementation of program GlueTray
 ********************************************************************)

PROGRAM _INIT

(* Glue Tray Man/Auto PB Colors *)
	HGW_2StatePB_0.BackColor_State0 := gBlue;
	HGW_2StatePB_0.ForeColor_State0 := gWhite;
	HGW_2StatePB_0.BackColor_State1 := gGreen;
	HGW_2StatePB_0.ForeColor_State1 := gBlack;

(* Glue Tray Slow Rotation PB Colors *)
	HGW_2StatePB_1.BackColor_State0 := gBlue;
	HGW_2StatePB_1.ForeColor_State0 := gWhite;
	HGW_2StatePB_1.BackColor_State1 := gGreen;
	HGW_2StatePB_1.ForeColor_State1 := gBlack;

END_PROGRAM
```

#### GlueTray.var - Local variables
```iecst
(********************************************************************
 * COPYRIGHT -- Microsoft
 ********************************************************************
 * Program: GlueTray
 * File: GlueTray.var
 * Author: pkiel
 * Created: July 19, 2011
 ********************************************************************
 * Local variables of program GlueTray
 ********************************************************************)
VAR
	GlueTray_Auto : BOOL;
	GlueTray_PB : BOOL;
	GlueTrayColor_Ind : UINT;
	GlueTraySR_On : BOOL;
	GlueTraySR_PB : BOOL;
	GlueTraySRColor_Ind : UINT;
	GlueTraySRText_Ind : UINT;
	GlueTrayText_Ind : UINT;
END_VAR
VAR RETAIN
	HGW_2StatePB_0 : HGW_2StatePB;
	HGW_2StatePB_1 : HGW_2StatePB;
END_VAR
```

### Program Logical/BagMachine_Section/Vacuum (IEC) - Former Vacuum control

#### VacuumCyclic.st
```iecst
(********************************************************************
 * COPYRIGHT -- Microsoft
 ********************************************************************
 * Program: Vacuum
 * File: VacuumCyclic.st
 * Author: pkiel
 * Created: July 19, 2011
 ********************************************************************
 * Implementation of program Vacuum
 ********************************************************************)

PROGRAM _CYCLIC

(* Vacuum Off/On From HMI *)
  HGW_2StatePB_0.PB := EDGEPOS(Vacuum_PB);
  VacuumText_Ind := HGW_2StatePB_0.Text_Ind;
  VacuumColor_Ind := HGW_2StatePB_0.Color_Ind;
  Vacuum_On := HGW_2StatePB_0.State1;
  HGW_2StatePB_0();

  (* Vacuum Control *)
  IF (Vacuum_On AND gI_SafetyRelay_EStopOK AND gQ_CR_MainPowerOn) THEN
    gQ_CON_Vacuum := 1;
  ELSE
    gQ_CON_Vacuum := 0;
  END_IF

END_PROGRAM
```

### Program Logical/BagMachine_Section/ExitTable (IEC) - Exit table control

#### ExitTable.var
```iecst
(********************************************************************
 * COPYRIGHT -- .
 ********************************************************************
 * Program: ExitTable
 * File: ExitTable.var
 * Author: dominique
 * Created: October 20, 2011
 ********************************************************************
 * Local variables of program ExitTable
 ********************************************************************)

VAR
  HMI_ExTb_rSPSlope            : REAL ;
  HMI_ExTb_bExitTableFaster_PB : BOOL ;
  HMI_ExTb_bExitTableSlower_PB : BOOL ;

  rIncrChangeSlope        : REAL ; (*Increment change slope, in %/(Bag/min)*)
  rIncrSlopeContinuChange : REAL ; (*Increment continually change, in (%/(Bag/min))/cycle*)
  rFactMulIncr            : REAL ;
  rCMD_RS_ExitTableSpeed  : REAL ;
  iCMD_Offset             : INT ;
  bFasterReq   : BOOL ;
  bSlowerReq   : BOOL ;
  bFastSlowReq : BOOL ;
  iMemoTime    : INT ;
  iDiffTime    : INT ;
  rDiffTime    : REAL ;
  stTON_ContinuChangeSlope_0 : TON ;
  stTON_ContinuChangeSlope_1 : TON ;
END_VAR

VAR CONSTANT

END_VAR
```

#### TableCyclic.st
```iecst
(********************************************************************
 * COPYRIGHT -- .
 ********************************************************************
 * Program: ExitTable
 * File: TableCyclic.st
 * Author: dominique
 * Created: October 20, 2011
 ********************************************************************
 * Implementation of program ExitTable
 ********************************************************************)

PROGRAM _CYCLIC

    bFasterReq := gI_SS_ExitTableFaster OR HMI_ExTb_bExitTableFaster_PB ;
    bSlowerReq := gI_SS_ExitTableSlower OR HMI_ExTb_bExitTableSlower_PB ;
    bFastSlowReq := bFasterReq OR bSlowerReq ;

    // Change slope by increment
    IF EDGEPOS(bFasterReq) THEN
      gRecipeActive.rSlopeExitTable := gRecipeActive.rSlopeExitTable + rIncrChangeSlope ;
    END_IF ;
    IF EDGEPOS(bSlowerReq) THEN
      gRecipeActive.rSlopeExitTable := gRecipeActive.rSlopeExitTable - rIncrChangeSlope ;
    END_IF ;

    // Change continually slope after 1s
    stTON_ContinuChangeSlope_0(IN:=bFastSlowReq, PT:=T#1s) ;
    // Change faster after 3s
    stTON_ContinuChangeSlope_0(IN:=bFastSlowReq, PT:=T#3s) ;
    IF stTON_ContinuChangeSlope_0.Q THEN
      rFactMulIncr := 1.0 ;
    END_IF ;
    IF stTON_ContinuChangeSlope_1.Q THEN
      rFactMulIncr := 6.0 ;
    END_IF ;
    IF bFasterReq THEN
      gRecipeActive.rSlopeExitTable := gRecipeActive.rSlopeExitTable + rIncrSlopeContinuChange * rFactMulIncr ;
    END_IF ;
    IF bSlowerReq THEN
      gRecipeActive.rSlopeExitTable := gRecipeActive.rSlopeExitTable - rIncrSlopeContinuChange * rFactMulIncr ;
    END_IF ;

    // Limit
    gRecipeActive.rSlopeExitTable := LIMIT(0,gRecipeActive.rSlopeExitTable,400) ;

    // Actual Speed Exit Table calculation
    // With gRecipeActive.rSlopeExitTable = 100% the maximum speed of the green belts on the exit table is reached when machine runs at maximum speed in bag/min
    rCMD_RS_ExitTableSpeed := gRecipeActive.rSlopeExitTable/100 * gActualMachineSpeed_BPM/gr_rMachMaxSpeed_BPM ;
    rCMD_RS_ExitTableSpeed := LIMIT(0,rCMD_RS_ExitTableSpeed,1.0) ;

    gQ_CMD_RS_ExitTableSpeed := REAL_TO_INT(rCMD_RS_ExitTableSpeed * C_rMaxAna) + iCMD_Offset ;

END_PROGRAM
```

#### TableInit.st
```iecst
(********************************************************************
 * COPYRIGHT -- .
 ********************************************************************
 * Program: ExitTable
 * File: TableInit.st
 * Author: dominique
 * Created: October 20, 2011
 ********************************************************************
 * Implementation of program ExitTable
 ********************************************************************)

PROGRAM _INIT

    rIncrChangeSlope        := 1.2 ;
    rIncrSlopeContinuChange := 0.1 ;

    iCMD_Offset := 1200 ;

END_PROGRAM
```

### Program Logical/BagMachine_Section/3Web_Unit (IEC) - 3Web_Unit control

#### 3Web_Unit.var - Local variables
```iecst
(********************************************************************
 * COPYRIGHT -- .
 ********************************************************************
 * Program: 3Web_Unit
 * File: 3Web_Unit.var
 * Author: dominique
 * Created: November 05, 2011
 ********************************************************************
 * Local variables of program 3Web_Unit
 ********************************************************************)

VAR
  HMI_bDeflectorFanOnOff_PB : BOOL;
  bDeflectorFan_On        : BOOL;
  uiDeflectorFanColor_Ind : UINT;
  uiDeflectorFanText_Ind  : UINT;
END_VAR
VAR RETAIN
  HGW_2StatePB_0 : HGW_2StatePB;
END_VAR
```

### Program Logical/BagMachine_Section/GlobProgCalc (IEC) - Global program calculation

#### GlobProgCalcInit.st
```iecst
(********************************************************************
 * COPYRIGHT -- .
 ********************************************************************
 * Program: GlobProgCalc
 * File: GlobProgCalcInit.st
 * Author: dominique
 * Created: October 27, 2011
 ********************************************************************
 * Implementation of program GlobProgCalc
 ********************************************************************)

PROGRAM _INIT

    // Init g_rNumbPliers because used in division
    rRepeatMetric := gRecipeActive.Repeat*25.4;
    IF (rRepeatMetric > gr_rBagSize4_2Pliers_mm) THEN
      g_rNumbPliers := 2.0 ;
    ELSE
      g_rNumbPliers := 4.0 ;
    END_IF ;

  // Bag size limite
  g_rMaxBagSize_RS15_mm := 400.0 ;
  g_rMinBagSize_RS15_mm := 105.0 ;
  g_rMaxBagSize_RS26_mm := 760.0 ;
  g_rMinBagSize_RS26_mm := 160.0 ;
  g_rMaxBagSize_EnvB_mm := 760.0 ;
  g_rMinBagSize_EnvB_mm := 240.0 ;

// -----------------------------------------------------------------------------
    // Machine devices activation  RS15_RX_30005

    // Machie Type
    g_iMachType := C_iRS15 ;

    // Glue RS
    gRecipeActive.bSelTypeRSGlue := 0 ; // D.M. 22/08/2012 Only Cold Glue for this machine RS15_RX_30005

    // Unwinder
    g_bUnwindInMach := 1 ;
    g_bUnwindEndRelPapInMach := 1 ;
    g_bUnwindEndRelPolyInMach := 0 ;

    // 3Web unit
    g_b3WebUnitInMach := 0 ;

    // FP_Dryer unit
    g_bDryerInMach   := 1 ;
    g_bHeatDryInMach := 1 ;

    // Flexo Press in machine
    gA[2].bInMach := 1 ;

    // Cold Micro Perf in machine
    gA[8].bInMach := 0 ;

    // Envelope Bag in machine
    gA[12].bInMach := 0 ;
    gA[13].bInMach := 0 ;

    // Hot Micro Perf in machine
    gA[15].bInMach := 0 ;

END_PROGRAM
```

### Program Logical/SupervisoryControl_Section/Alarm_Section/EStopReset (IEC) - E-Stop Relay and Alarm Reset

#### EStopResetCyclic.ld
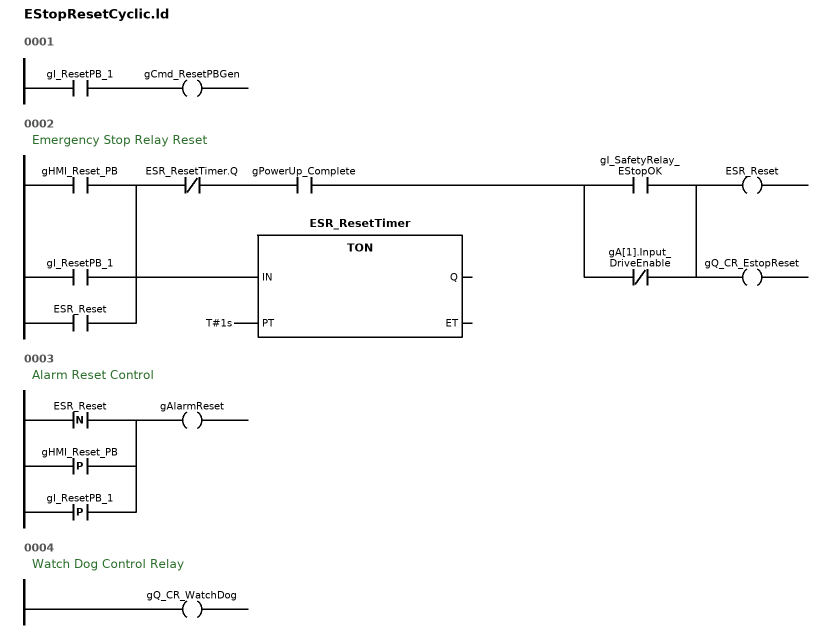
Ladder, written as Structured Text:
```iecst
(********************************************************************
 * COPYRIGHT --
 ********************************************************************
 * Program: EStopReset
 * File: EStopResetCyclic.ld
 * Author: pkiel
 * Created: October 12, 2009
 ********************************************************************
 * Implementation of program EStopReset
 ********************************************************************)

PROGRAM _CYCLIC
VAR
    _p1 : BOOL;
    _p2 : BOOL;
    _e3 : F_TRIG;
    _e4 : R_TRIG;
    _e5 : R_TRIG;
END_VAR
(* Network 1 *)
gCmd_ResetPBGen := gI_ResetPB_1;

(* Network 2: Emergency Stop Relay Reset *)
_p1 := (gHMI_Reset_PB OR gI_ResetPB_1 OR ESR_Reset) AND NOT ESR_ResetTimer.Q AND gPowerUp_Complete;
_p2 := ESR_Reset;
ESR_Reset := _p1 AND (gI_SafetyRelay_EStopOK OR NOT gA[1].Input_DriveEnable);
ESR_ResetTimer(IN := gHMI_Reset_PB OR gI_ResetPB_1 OR _p2, PT := T#1s);
gQ_CR_EstopReset := _p1 AND (gI_SafetyRelay_EStopOK OR NOT gA[1].Input_DriveEnable);

(* Network 3: Alarm Reset Control *)
_e3(CLK := ESR_Reset);
_e4(CLK := gHMI_Reset_PB);
_e5(CLK := gI_ResetPB_1);
gAlarmReset := _e3.Q OR _e4.Q OR _e5.Q;

(* Network 4: Watch Dog Control Relay *)
gQ_CR_WatchDog := TRUE;
END_PROGRAM
```

### Program Logical/SupervisoryControl_Section/Alarm_Section/Alarms1 (IEC) - Bag Machine Alarm Monitoring

#### actAnimAlarmVisu.st
```iecst
(********************************************************************
 * COPYRIGHT -- .
 ********************************************************************
 * Program: Alarms1
 * File: actAnimAlarmVisu.st
 * Author: dominique
 * Created: January 27, 2012
 ********************************************************************
 * Implementation of program Alarms1
 ********************************************************************)

(*Alarme animation on visu*)
ACTION actAnimAlarmVisu:

  H_FB_Flash_0(IN_bEnable:=1, IN_rNumFlashPerSec:=1.0) ;

  // BP AU Panel +R4
  IF gI_EstopPB_1            AND
     H_FB_Flash_0.OUT_bFlash THEN
    iVisiblES_BP1 := 0 ; // Visible
  ELSE
    iVisiblES_BP1 := 1 ; // Unvisible
  END_IF
  // BP AU Panel +R3
  IF gI_EstopPB_2            AND
     H_FB_Flash_0.OUT_bFlash THEN
    iVisiblES_BP2 := 0 ; // Visible
  ELSE
    iVisiblES_BP2 := 1 ; // Unvisible
  END_IF
  // BP AU Panel +R1
  IF gI_EstopPB_3            AND
     H_FB_Flash_0.OUT_bFlash THEN
    iVisiblES_BP3 := 0 ; // Visible
  ELSE
    iVisiblES_BP3 := 1 ; // Unvisible
  END_IF
  // BP AU Panel +R3
  IF gI_EstopPB_4            AND
     H_FB_Flash_0.OUT_bFlash THEN
    iVisiblES_BP4 := 0 ; // Visible
  ELSE
    iVisiblES_BP4 := 1 ; // Unvisible
  END_IF
  // BP AU Panel +R1A
  IF gI_EstopPB_5            AND
     H_FB_Flash_0.OUT_bFlash THEN
    iVisiblES_BP5 := 0 ; // Visible
  ELSE
    iVisiblES_BP5 := 1 ; // Unvisible
  END_IF
  // BP AU Footswitch Jog
  IF NOT(gI_SafetyRelay_EStopOK) AND
     gI_JogPB_1                  AND
     H_FB_Flash_0.OUT_bFlash     THEN
    iVisiblES_BP6 := 0 ; // Visible
  ELSE
    iVisiblES_BP6 := 1 ; // Unvisible
  END_IF

  // BP AU Flexo
  IF gI_EstopPB_FlexoPress   AND
    H_FB_Flash_0.OUT_bFlash THEN
    iVisiblES_BP9 := 0 ; // Visible
  ELSE
    iVisiblES_BP9 := 1 ; // Unvisible
  END_IF

  // BP AU DHS
  IF gI_EstopPB_Unwind       AND
    H_FB_Flash_0.OUT_bFlash THEN
    iVisiblES_BP10 := 0 ; // Visible
  ELSE
    iVisiblES_BP10 := 1 ; // Unvisible
  END_IF

END_ACTION
```

#### actIO_Ex_FailDetect_E1_L3.st
```iecst
(********************************************************************
 * COPYRIGHT -- .
 ********************************************************************
 * Program: Alarms1
 * File: actIO_Ex_FailDetect.st
 * Author: dominique
 * Created: October 16, 2011
 ********************************************************************
 * Implementation of program Alarms1
 ********************************************************************)

ACTION actIO_Ex_FailDetect_E1_L3 :
//ACTION for calculation failures of REM_IO_Ex modules

  // ----------------------------------------------------------------------------------------------------------------------------------------------------------
  // Detection failures of REM_IO_E1 modules
  FOR iIndex := 1 TO C_iMaxAlmIO_E1 DO
    IF NOT(stModuleOK_IO_E1_Slot[iIndex].bStat) THEN
      bAlarmIO_E1[iIndex] := 1 ;
    END_IF
    IF stModuleOK_IO_E1_Slot[iIndex].bStat AND
       gAlarmReset                         THEN
      bAlarmIO_E1[iIndex] := 0 ;
    END_IF
    IF iIndex>C_iNumBefFirstIO_E1+C_iNumDI_E1+C_iNumAI_E1+1+C_iNumDO_E1+C_iNumAO_E1 THEN
      bAlarmIO_E1[iIndex] := 0 ;
    END_IF
  END_FOR ;

  // Module type REM_IO_E1
  // PowerLink Head module
  stModuleOK_IO_E1_Slot[1].strType := 'X20BC0083' ;
  // Alim module
  stModuleOK_IO_E1_Slot[2].strType := 'X20PS9400' ;
  // DI modules
  FOR iIndex := 1+C_iNumBefFirstIO_E1 TO C_iNumDI_E1+C_iNumBefFirstIO_E1 DO
    stModuleOK_IO_E1_Slot[iIndex].strType := 'X20DI9371' ;
  END_FOR ;
  // AI modules
  IF (C_iNumAI_E1>0) THEN
    FOR iIndex := 1+C_iNumBefFirstIO_E1+C_iNumDI_E1 TO C_iNumBefFirstIO_E1+C_iNumDI_E1+C_iNumAI_E1 DO
      //stModuleOK_IO_E1_Slot[iIndex].strType := 'X20AI2622' ;
      stModuleOK_IO_E1_Slot[iIndex].strType := 'X20AT2222' ;
    END_FOR ;
  END_IF
  // Output alim module
  stModuleOK_IO_E1_Slot[C_iNumBefFirstIO_E1+C_iNumDI_E1+C_iNumAI_E1+1].strType := 'X20PS3300' ;
  // DO modules
  IF (C_iNumDO_E1>0) THEN
    FOR iIndex := C_iNumBefFirstIO_E1+C_iNumDI_E1+C_iNumAI_E1+2 TO C_iNumBefFirstIO_E1+C_iNumDI_E1+C_iNumAI_E1+1+C_iNumDO_E1 DO // +1 et +2 because alim module
      stModuleOK_IO_E1_Slot[iIndex].strType := 'X20DO9322' ;
    END_FOR ;
  END_IF
  // AO modules
  IF (C_iNumAO_E1>0) THEN
    FOR iIndex := C_iNumBefFirstIO_E1+C_iNumDI_E1+C_iNumAI_E1+2+C_iNumDO_E1 TO C_iNumBefFirstIO_E1+C_iNumDI_E1+C_iNumAI_E1+1+C_iNumDO_E1+C_iNumAO_E1 DO
      stModuleOK_IO_E1_Slot[iIndex].strType := 'X20A02622' ;
    END_FOR ;
  END_IF
  // General alarme calculation
  bAlarmGenIO_E1 := bAlarmIO_E1[1]  OR
                    bAlarmIO_E1[2]  OR
                    bAlarmIO_E1[3]  OR
                    bAlarmIO_E1[4]  OR
                    bAlarmIO_E1[5]  OR
                    bAlarmIO_E1[6]  OR
                    bAlarmIO_E1[7]  OR
                    bAlarmIO_E1[8]  OR
                    bAlarmIO_E1[9]  OR
                    bAlarmIO_E1[10] OR
                    bAlarmIO_E1[11] OR
                    bAlarmIO_E1[12] OR
                    bAlarmIO_E1[13] OR
                    bAlarmIO_E1[14] OR
                    bAlarmIO_E1[15] OR
                    bAlarmIO_E1[16] OR
                    bAlarmIO_E1[17] OR
                    bAlarmIO_E1[18] OR
                    bAlarmIO_E1[19] OR
                    bAlarmIO_E1[20] ; //OR
                    (*bAlarmIO_E1[21] OR
                    bAlarmIO_E1[22] OR
                    bAlarmIO_E1[23] OR
                    bAlarmIO_E1[24] OR
                    bAlarmIO_E1[25] OR
                    bAlarmIO_E1[26] OR
                    bAlarmIO_E1[27] OR
                    bAlarmIO_E1[28] OR
                    bAlarmIO_E1[29] OR
                    bAlarmIO_E1[30] OR
                    bAlarmIO_E1[31] OR
                    bAlarmIO_E1[32] OR
                    bAlarmIO_E1[33] OR
                    bAlarmIO_E1[34] OR
                    bAlarmIO_E1[35] OR
                    bAlarmIO_E1[36] OR
                    bAlarmIO_E1[37] OR
                    bAlarmIO_E1[38] OR
                    bAlarmIO_E1[39] OR
                    bAlarmIO_E1[40] ;*)

  // ----------------------------------------------------------------------------------------------------------------------------------------------------------
  // Detection failures of REM_IO_L3 modules
  FOR iIndex := 1 TO C_iMaxAlmIO_L3 DO
    IF NOT(stModuleOK_IO_L3_Slot[iIndex].bStat) THEN
      bAlarmIO_L3[iIndex] := 1 ;
    END_IF
    IF stModuleOK_IO_L3_Slot[iIndex].bStat AND
       gAlarmReset                         THEN
      bAlarmIO_L3[iIndex] := 0 ;
    END_IF
    IF iIndex>C_iNumBefFirstIO_L3+C_iNumDI_L3+C_iNumAI_L3+1+C_iNumDO_L3+C_iNumAO_L3+C_iX2XExt_L3 THEN
      bAlarmIO_L3[iIndex] := 0 ;
    END_IF
  END_FOR ;
  // Module type REM_IO_L3
  // PowerLink Head module
  //stModuleOK_IO_L3_Slot[1].strType := 'X20BC0083' ;
  // Alim module
  //stModuleOK_IO_L3_Slot[2].strType := 'X20PS9400' ;
  // Alim module + PowerLink network
  stModuleOK_IO_L3_Slot[1].strType := 'X20BR9300' ;
  // DI modules
  FOR iIndex := 1+C_iNumBefFirstIO_L3 TO C_iNumBefFirstIO_L3+C_iNumDI_L3 DO
    stModuleOK_IO_L3_Slot[iIndex].strType := 'X20DI9371' ;
  END_FOR ;
  // AI modules
  IF (C_iNumAI_L3>0) THEN
    FOR iIndex := 1+C_iNumBefFirstIO_L3+C_iNumDI_L3 TO C_iNumBefFirstIO_L3+C_iNumDI_L3+C_iNumAI_L3 DO
      stModuleOK_IO_L3_Slot[iIndex].strType := 'X20AI2622' ;
    END_FOR ;
  END_IF
  // Output alim module
  stModuleOK_IO_L3_Slot[C_iNumBefFirstIO_L3+C_iNumDI_L3+C_iNumAI_L3+1].strType := 'X20PS3300' ;
  // DO modules
  IF (C_iNumDO_L3>0) THEN
    FOR iIndex := C_iNumBefFirstIO_L3+C_iNumDI_L3+C_iNumAI_L3+2 TO C_iNumBefFirstIO_L3+C_iNumDI_L3+C_iNumAI_L3+1+C_iNumDO_L3 DO // +2 et +1 because alim module
      stModuleOK_IO_L3_Slot[iIndex].strType := 'X20DO9322' ;
    END_FOR ;
  END_IF
  // AO modules
  IF (C_iNumAO_L3>0) THEN
    FOR iIndex := C_iNumBefFirstIO_L3+C_iNumDI_L3+C_iNumAI_L3+2+C_iNumDO_L3 TO C_iNumBefFirstIO_L3+C_iNumDI_L3+C_iNumAI_L3+1+C_iNumDO_L3+C_iNumAO_L3 DO
      stModuleOK_IO_L3_Slot[iIndex].strType := 'X20A02622' ;
    END_FOR ;
  END_IF
  // Bus X2X Output module
  stModuleOK_IO_L3_Slot[C_iNumBefFirstIO_L3+C_iNumDI_L3+C_iNumAI_L3+1+C_iNumDO_L3+C_iNumAO_L3+1].strType := 'X20BT9100' ;

  // General alarme calculation
  bAlarmGenIO_L3 := bAlarmIO_L3[1]  OR
                    bAlarmIO_L3[2]  OR
                    bAlarmIO_L3[3]  OR
                    bAlarmIO_L3[4]  OR
                    bAlarmIO_L3[5]  OR
                    bAlarmIO_L3[6]  OR
                    bAlarmIO_L3[7]  OR
                    bAlarmIO_L3[8]  OR
                    bAlarmIO_L3[9]  OR
                    bAlarmIO_L3[10] OR
                    bAlarmIO_L3[11] OR
                    bAlarmIO_L3[12] OR
                    bAlarmIO_L3[13] OR
                    bAlarmIO_L3[14] OR
                    bAlarmIO_L3[15] OR
                    bAlarmIO_L3[16] OR
                    bAlarmIO_L3[17] OR
                    bAlarmIO_L3[18] OR
                    bAlarmIO_L3[19] OR
                    bAlarmIO_L3[20] ; //OR
                    (*bAlarmIO_L3[21] OR
                    bAlarmIO_L3[22] OR
                    bAlarmIO_L3[23] OR
                    bAlarmIO_L3[24] OR
                    bAlarmIO_L3[25] OR
                    bAlarmIO_L3[26] OR
                    bAlarmIO_L3[27] OR
                    bAlarmIO_L3[28] OR
                    bAlarmIO_L3[29] OR
                    bAlarmIO_L3[30] OR
                    bAlarmIO_L3[31] OR
                    bAlarmIO_L3[32] OR
                    bAlarmIO_L3[33] OR
                    bAlarmIO_L3[34] OR
                    bAlarmIO_L3[35] OR
                    bAlarmIO_L3[36] OR
                    bAlarmIO_L3[37] OR
                    bAlarmIO_L3[38] OR
                    bAlarmIO_L3[39] OR
                    bAlarmIO_L3[40] ;*)

END_ACTION
```

#### actIO_Ex_FailDetect_L15.st
```iecst
(********************************************************************
 * COPYRIGHT -- .
 ********************************************************************
 * Program: Alarms1
 * File: actIO_Ex_FailDetect.st
 * Author: dominique
 * Created: October 16, 2011
 ********************************************************************
 * Implementation of program Alarms1
 ********************************************************************)

ACTION actIO_Ex_FailDetect_L15 :
//ACTION for calculation failures of REM_IO_Ex modules

  // ----------------------------------------------------------------------------------------------------------------------------------------------------------
  // Detection failures of REM_IO_L15 modules
  FOR iIndex := 1 TO C_iMaxAlmIO_L15 DO
    IF NOT(stModuleOK_IO_L15_Slot[iIndex].bStat) THEN
      bAlarmIO_L15[iIndex] := g_bIndSelBundProd ;
    END_IF
    IF ( stModuleOK_IO_L15_Slot[iIndex].bStat OR
         NOT(gA[15].bInMach) )                AND
       gAlarmReset                            THEN
      bAlarmIO_L15[iIndex] := 0 ;
    END_IF
    IF iIndex>C_iNumBefFirstIO_L15+C_iNumDI_L15+C_iNumAI_L15+1+C_iNumDO_L15+C_iNumAO_L15+C_iX2XExt_L15 THEN
      bAlarmIO_L15[iIndex] := 0 ;
    END_IF
  END_FOR ;
  // Module type REM_IO_L15
  // PowerLink Head module
  //stModuleOK_IO_L15_Slot[1].strType := 'X20BC0083' ;
  // Alim module
  //stModuleOK_IO_L15_Slot[2].strType := 'X20PS9400' ;
  // Alim module + PowerLink network
  stModuleOK_IO_L15_Slot[1].strType := 'X20BR9300' ;
  // DI modules
  FOR iIndex := 1+C_iNumBefFirstIO_L15 TO C_iNumDI_L15 DO
    stModuleOK_IO_L15_Slot[iIndex].strType := 'X20DI4371' ;
  END_FOR ;
  // AI modules
  IF (C_iNumAI_L15>0) THEN
    FOR iIndex := 1+C_iNumBefFirstIO_L15+C_iNumDI_L15 TO C_iNumBefFirstIO_L15+C_iNumDI_L15+C_iNumAI_L15 DO
      stModuleOK_IO_L15_Slot[iIndex].strType := 'X20AI2622' ;
    END_FOR ;
  END_IF
  // Output alim module
  //stModuleOK_IO_L15_Slot[C_iNumBefFirstIO_L15+C_iNumDI_L15+C_iNumAI_L15+1].strType := 'X20PS3300' ;
  stModuleOK_IO_L15_Slot[C_iNumBefFirstIO_L15+C_iNumDI_L15+C_iNumAI_L15+1].strType := 'X20PS2100' ;
  // DO modules
  IF (C_iNumDO_L15>0) THEN
    FOR iIndex := C_iNumBefFirstIO_L15+C_iNumDI_L15+C_iNumAI_L15+2 TO C_iNumBefFirstIO_L15+C_iNumDI_L15+C_iNumAI_L15+2+C_iNumDO_L15 DO // +2 because alim module
      stModuleOK_IO_L15_Slot[iIndex].strType := 'X20DO4322' ;
    END_FOR ;
  END_IF
  // AO modules
  IF (C_iNumAO_L15>0) THEN
    FOR iIndex := C_iNumBefFirstIO_L15+C_iNumDI_L15+C_iNumAI_L15+2+C_iNumDO_L15 TO C_iNumBefFirstIO_L15+C_iNumDI_L15+C_iNumAI_L15+2+C_iNumDO_L15+C_iNumAO_L15 DO
      stModuleOK_IO_L15_Slot[iIndex].strType := 'X20A02622' ;
    END_FOR ;
  END_IF
  // General alarme calculation
  bAlarmGenIO_L15 := bAlarmIO_L15[1]  OR
                    bAlarmIO_L15[2]  OR
                    bAlarmIO_L15[3]  OR
                    bAlarmIO_L15[4]  OR
                    bAlarmIO_L15[5]  OR
                    bAlarmIO_L15[6]  OR
                    bAlarmIO_L15[7]  OR
                    bAlarmIO_L15[8]  OR
                    bAlarmIO_L15[9]  OR
                    bAlarmIO_L15[10] OR
                    bAlarmIO_L15[11] OR
                    bAlarmIO_L15[12] OR
                    bAlarmIO_L15[13] OR
                    bAlarmIO_L15[14] OR
                    bAlarmIO_L15[15] OR
                    bAlarmIO_L15[16] OR
                    bAlarmIO_L15[17] OR
                    bAlarmIO_L15[18] OR
                    bAlarmIO_L15[19] OR
                    bAlarmIO_L15[20] ; //OR
                    (*bAlarmIO_L15[21] OR
                    bAlarmIO_L15[22] OR
                    bAlarmIO_L15[23] OR
                    bAlarmIO_L15[24] OR
                    bAlarmIO_L15[25] OR
                    bAlarmIO_L15[26] OR
                    bAlarmIO_L15[27] OR
                    bAlarmIO_L15[28] OR
                    bAlarmIO_L15[29] OR
                    bAlarmIO_L15[30] OR
                    bAlarmIO_L15[31] OR
                    bAlarmIO_L15[32] OR
                    bAlarmIO_L15[33] OR
                    bAlarmIO_L15[34] OR
                    bAlarmIO_L15[35] OR
                    bAlarmIO_L15[36] OR
                    bAlarmIO_L15[37] OR
                    bAlarmIO_L15[38] OR
                    bAlarmIO_L15[39] OR
                    bAlarmIO_L15[40] ;*)

END_ACTION
```

#### actIO_Ex_FailDetect_L9.st
```iecst
(********************************************************************
 * COPYRIGHT -- .
 ********************************************************************
 * Program: Alarms1
 * File: actIO_Ex_FailDetect.st
 * Author: dominique
 * Created: October 16, 2011
 ********************************************************************
 * Implementation of program Alarms1
 ********************************************************************)

ACTION actIO_Ex_FailDetect_L9 :
//ACTION for calculation failures of REM_IO_Ex modules

  // ----------------------------------------------------------------------------------------------------------------------------------------------------------
  // Detection failures of REM_IO_L9 modules
  FOR iIndex := 1 TO C_iMaxAlmIO_L9 DO
    IF NOT(stModuleOK_IO_L9_Slot[iIndex].bStat) THEN
      bAlarmIO_L9[iIndex] := g_bIndSelBundProd ;
    END_IF
    IF (stModuleOK_IO_L9_Slot[iIndex].bStat OR
        NOT(g_bIndSelBundProd))             AND
       gAlarmReset                          THEN
      bAlarmIO_L9[iIndex] := 0 ;
    END_IF
    IF iIndex>C_iNumBefFirstIO_L9+C_iNumDI_L9+C_iNumAI_L9+1+C_iNumDO_L9+C_iNumAO_L9+C_iX2XExt_L9 THEN
      bAlarmIO_L9[iIndex] := 0 ;
    END_IF
  END_FOR ;

  // Module type REM_IO_L9
  // PowerLink Head module
  //stModuleOK_IO_L9_Slot[1].strType := 'X20BC0083' ;
  // Alim module
  //stModuleOK_IO_L9_Slot[2].strType := 'X20PS9400' ;
  // Alim module + PowerLink network
  stModuleOK_IO_L9_Slot[1].strType := 'X20BR9300' ;
  // DI modules
  FOR iIndex := 1+C_iNumBefFirstIO_L9 TO C_iNumBefFirstIO_L9+C_iNumDI_L9 DO
    stModuleOK_IO_L9_Slot[iIndex].strType := 'X20DI4371' ;
  END_FOR ;
  // AI modules
  IF (C_iNumAI_L9>0) THEN
    FOR iIndex := 1+C_iNumBefFirstIO_L9+C_iNumDI_L9 TO C_iNumBefFirstIO_L9+C_iNumDI_L9+C_iNumAI_L9 DO
      stModuleOK_IO_L9_Slot[iIndex].strType := 'X20AI2622' ;
    END_FOR ;
  END_IF
  // Output alim module
  stModuleOK_IO_L9_Slot[C_iNumBefFirstIO_L9+C_iNumDI_L9+C_iNumAI_L9+1].strType := 'X20PS3300' ;
  // DO modules
  IF (C_iNumDO_L9>0) THEN
    FOR iIndex := C_iNumBefFirstIO_L9+C_iNumDI_L9+C_iNumAI_L9+2 TO C_iNumBefFirstIO_L9+C_iNumDI_L9+C_iNumAI_L9+1+C_iNumDO_L9 DO // +1 et +2 because alim module
      stModuleOK_IO_L9_Slot[iIndex].strType := 'X20DO4322' ;
    END_FOR ;
  END_IF
  // AO modules
  IF (C_iNumAO_L9>0) THEN
    FOR iIndex := C_iNumBefFirstIO_L9+C_iNumDI_L9+C_iNumAI_L9+2+C_iNumDO_L9 TO C_iNumBefFirstIO_L9+C_iNumDI_L9+C_iNumAI_L9+1+C_iNumDO_L9+C_iNumAO_L9 DO
      stModuleOK_IO_L9_Slot[iIndex].strType := 'X20A02622' ;
    END_FOR ;
  END_IF
  // General alarme calculation
  bAlarmGenIO_L9 := bAlarmIO_L9[1]  OR
                    bAlarmIO_L9[2]  OR
                    bAlarmIO_L9[3]  OR
                    bAlarmIO_L9[4]  OR
                    bAlarmIO_L9[5]  OR
                    bAlarmIO_L9[6]  OR
                    bAlarmIO_L9[7]  OR
                    bAlarmIO_L9[8]  OR
                    bAlarmIO_L9[9]  OR
                    bAlarmIO_L9[10] OR
                    bAlarmIO_L9[11] OR
                    bAlarmIO_L9[12] OR
                    bAlarmIO_L9[13] OR
                    bAlarmIO_L9[14] OR
                    bAlarmIO_L9[15] OR
                    bAlarmIO_L9[16] OR
                    bAlarmIO_L9[17] OR
                    bAlarmIO_L9[18] OR
                    bAlarmIO_L9[19] OR
                    bAlarmIO_L9[20] ; //OR
                    (*bAlarmIO_L9[21] OR
                    bAlarmIO_L9[22] OR
                    bAlarmIO_L9[23] OR
                    bAlarmIO_L9[24] OR
                    bAlarmIO_L9[25] OR
                    bAlarmIO_L9[26] OR
                    bAlarmIO_L9[27] OR
                    bAlarmIO_L9[28] OR
                    bAlarmIO_L9[29] OR
                    bAlarmIO_L9[30] OR
                    bAlarmIO_L9[31] OR
                    bAlarmIO_L9[32] OR
                    bAlarmIO_L9[33] OR
                    bAlarmIO_L9[34] OR
                    bAlarmIO_L9[35] OR
                    bAlarmIO_L9[36] OR
                    bAlarmIO_L9[37] OR
                    bAlarmIO_L9[38] OR
                    bAlarmIO_L9[39] OR
                    bAlarmIO_L9[40] ;*)

END_ACTION
```

#### Alarms1Cyclic.ld
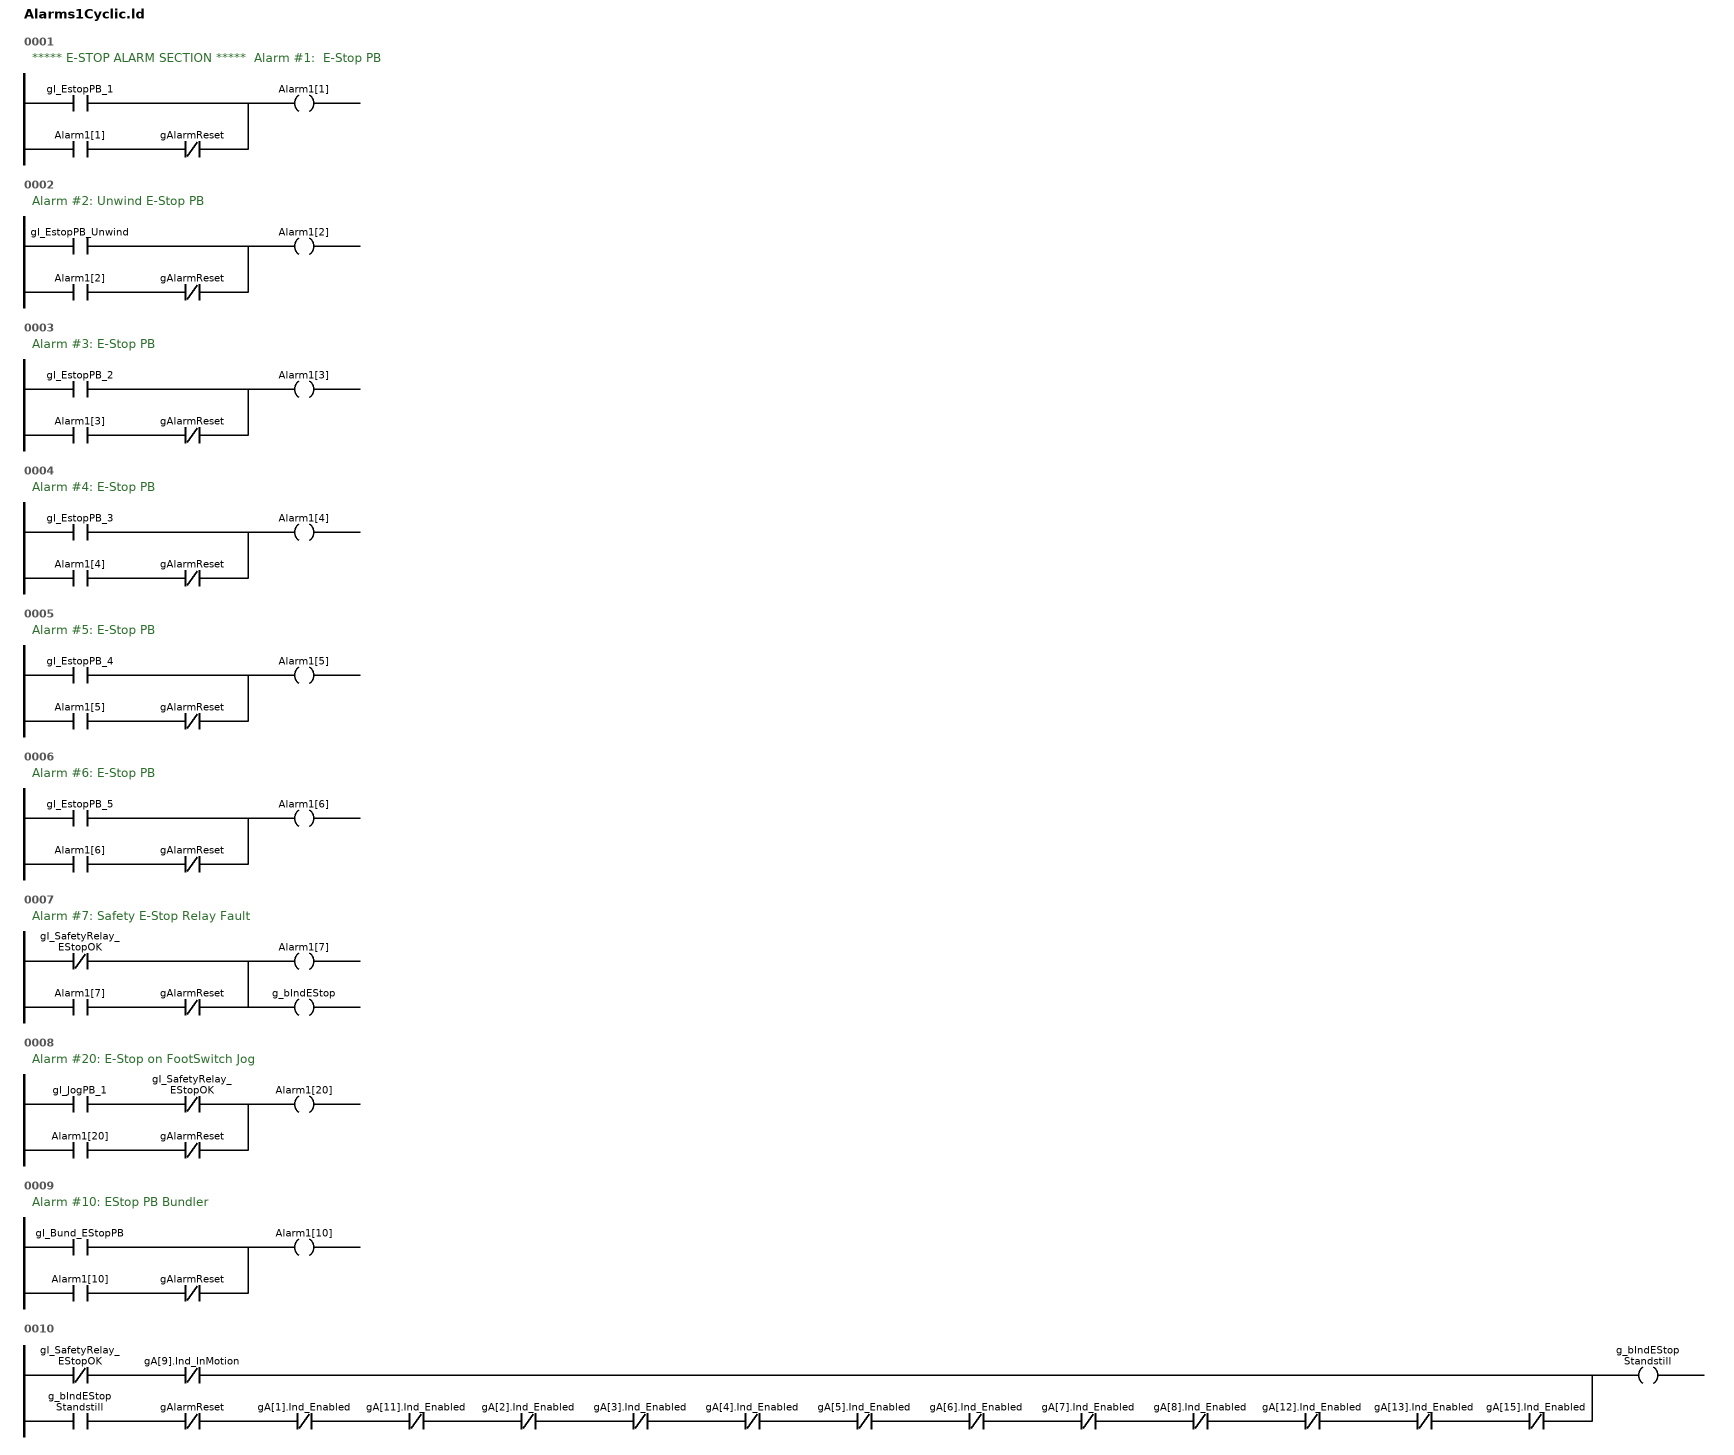
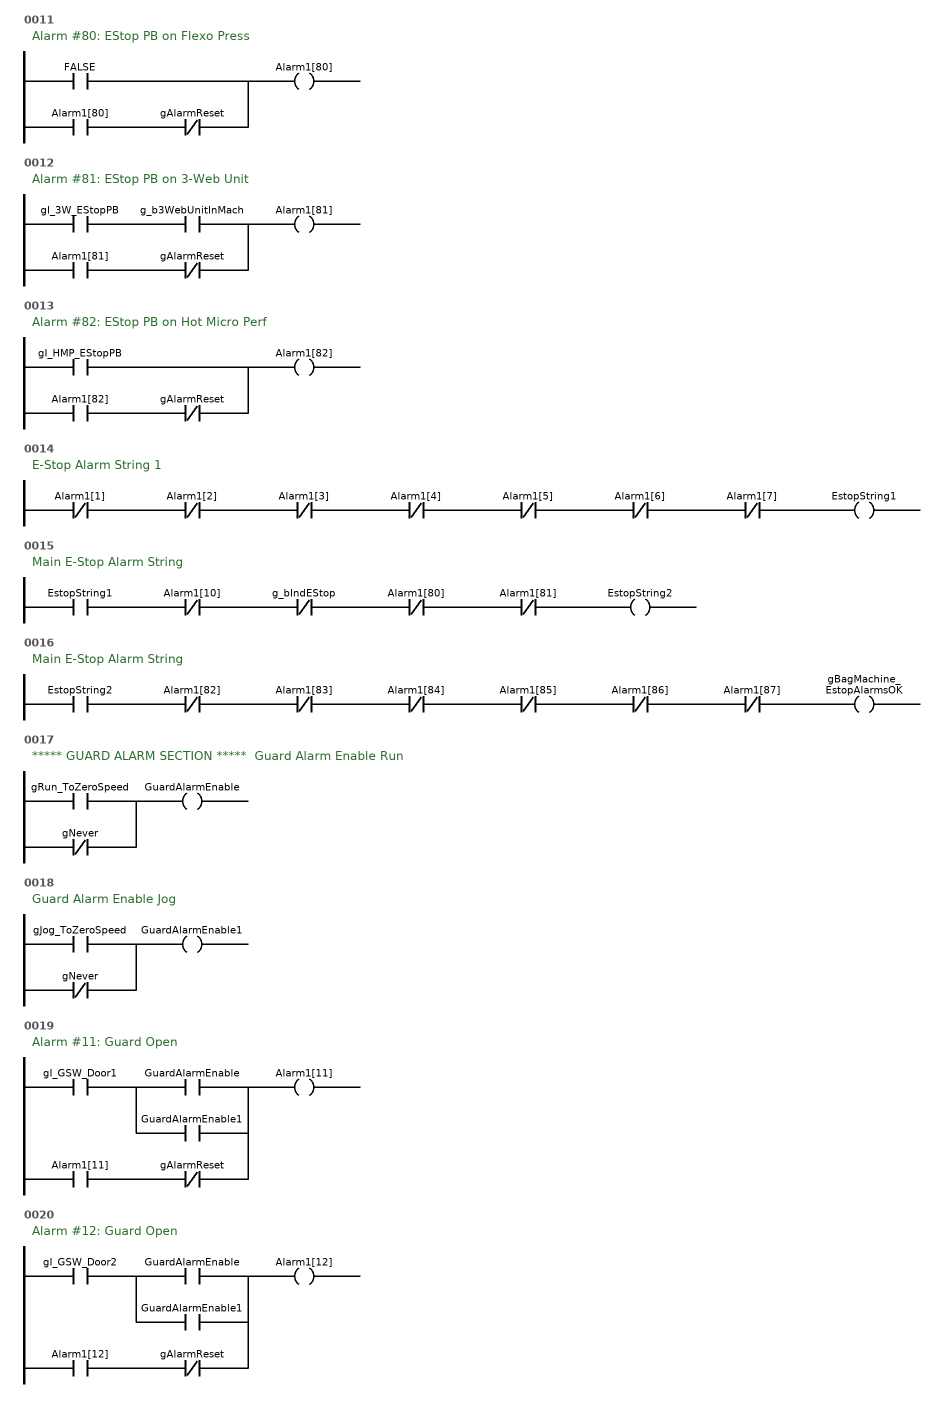
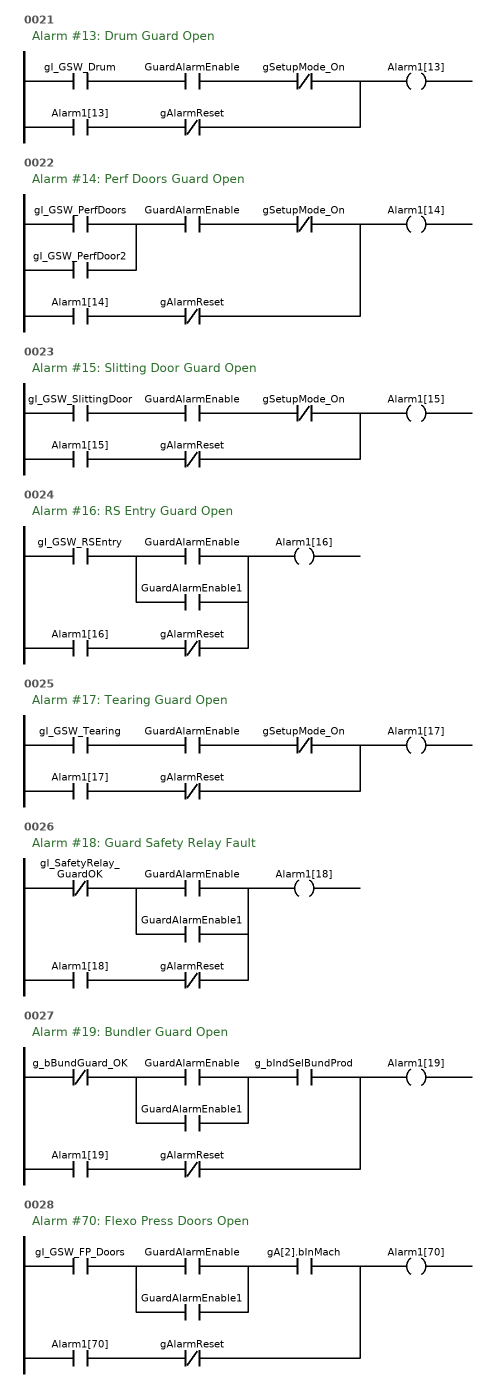
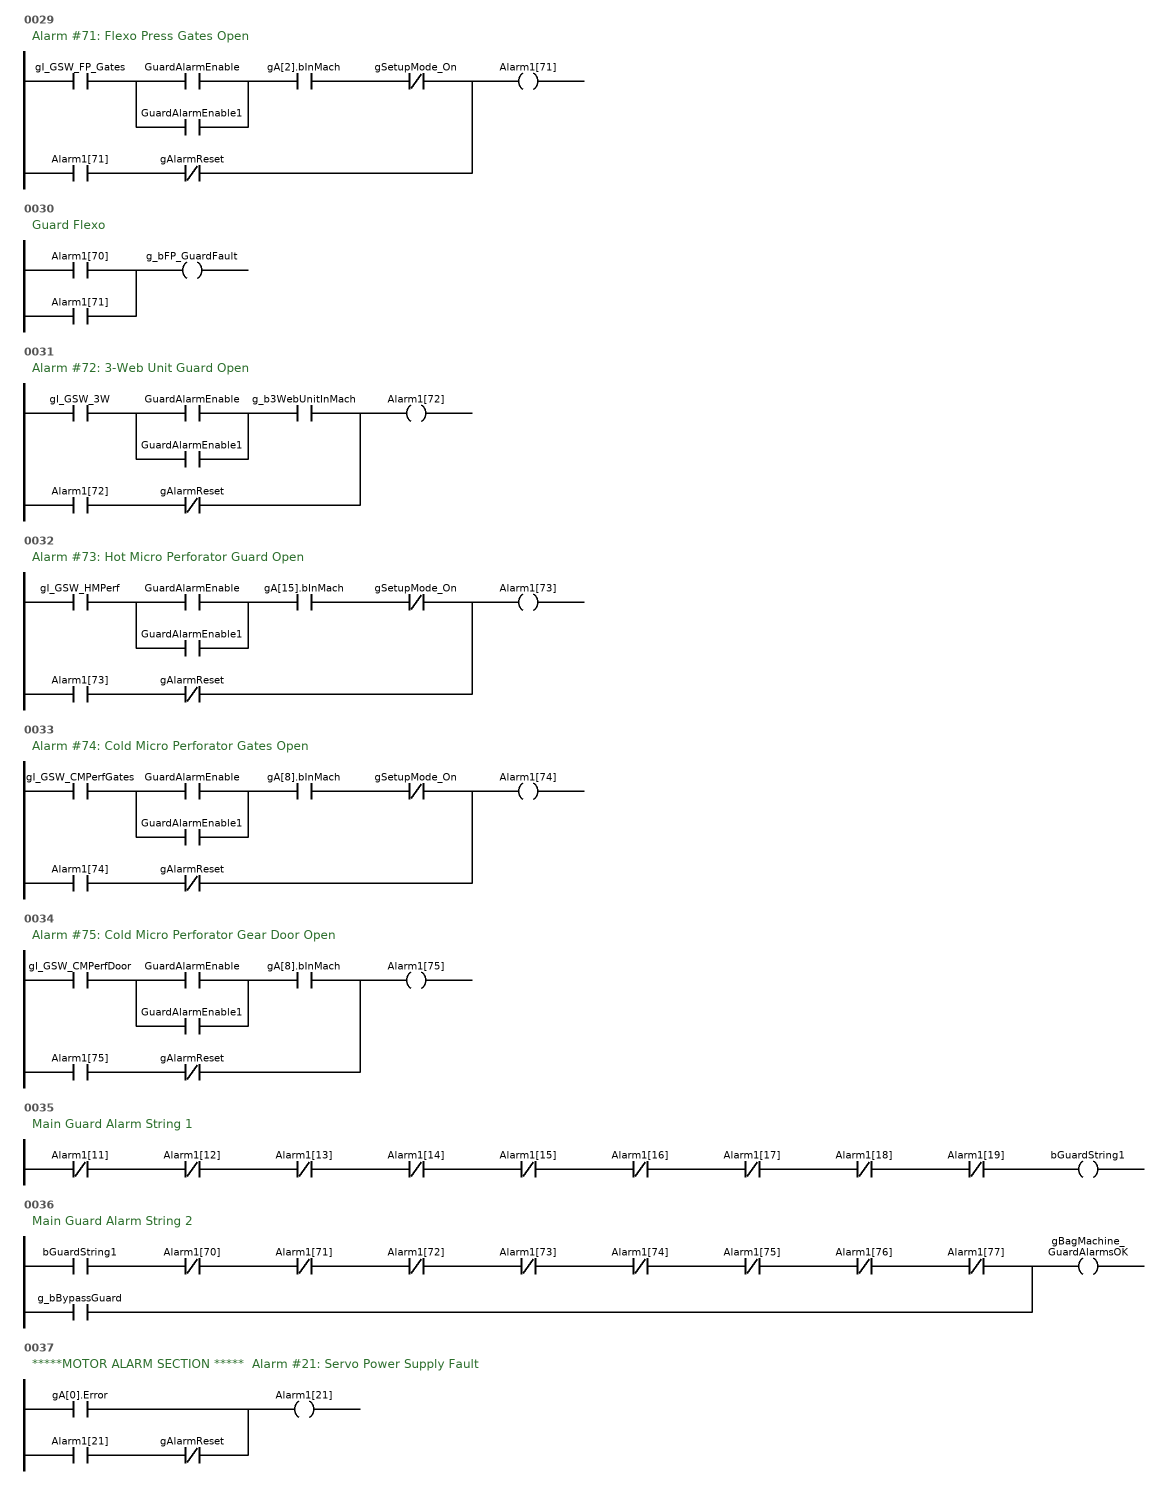
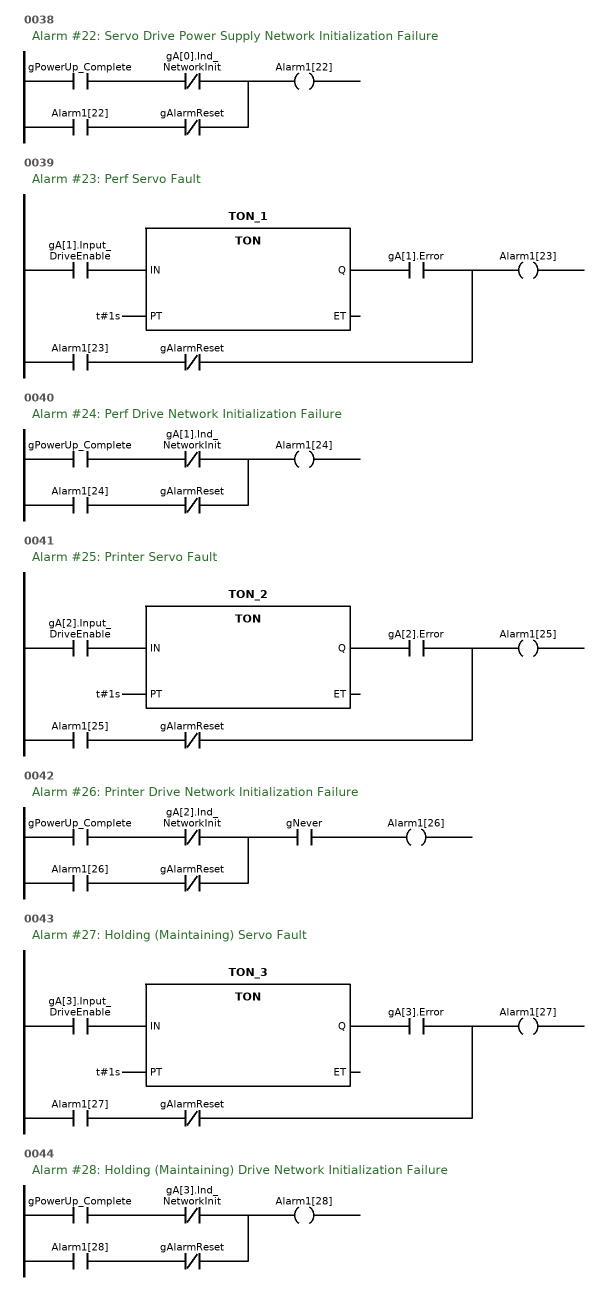
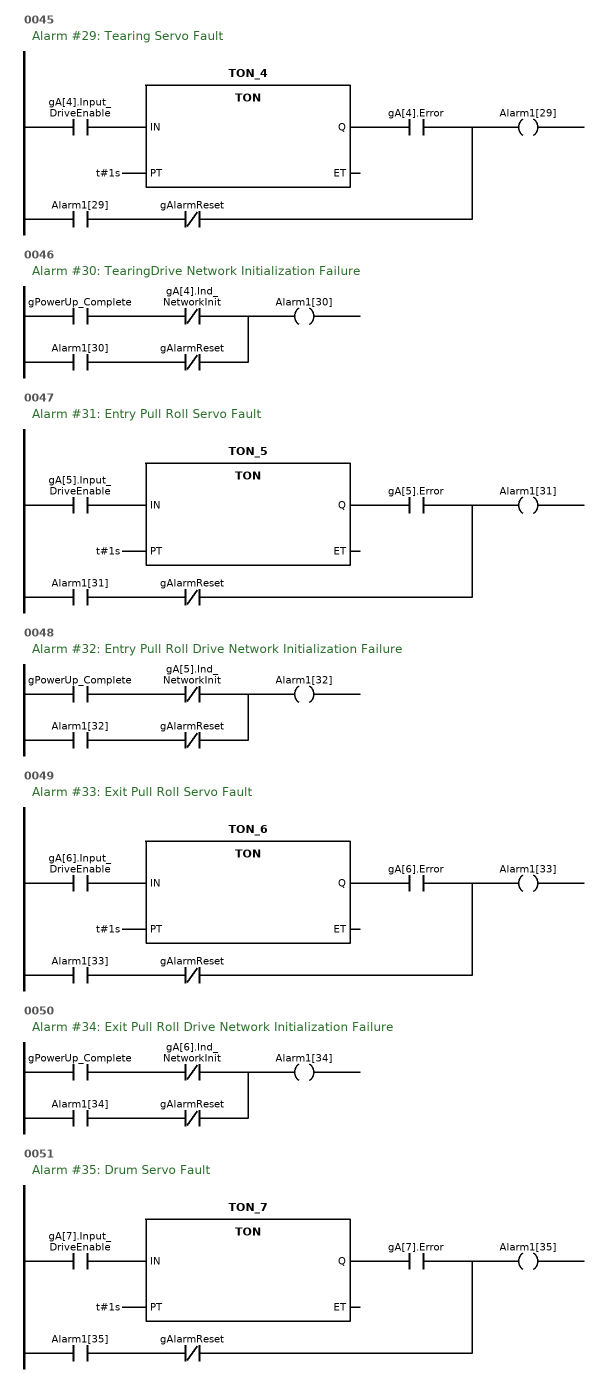
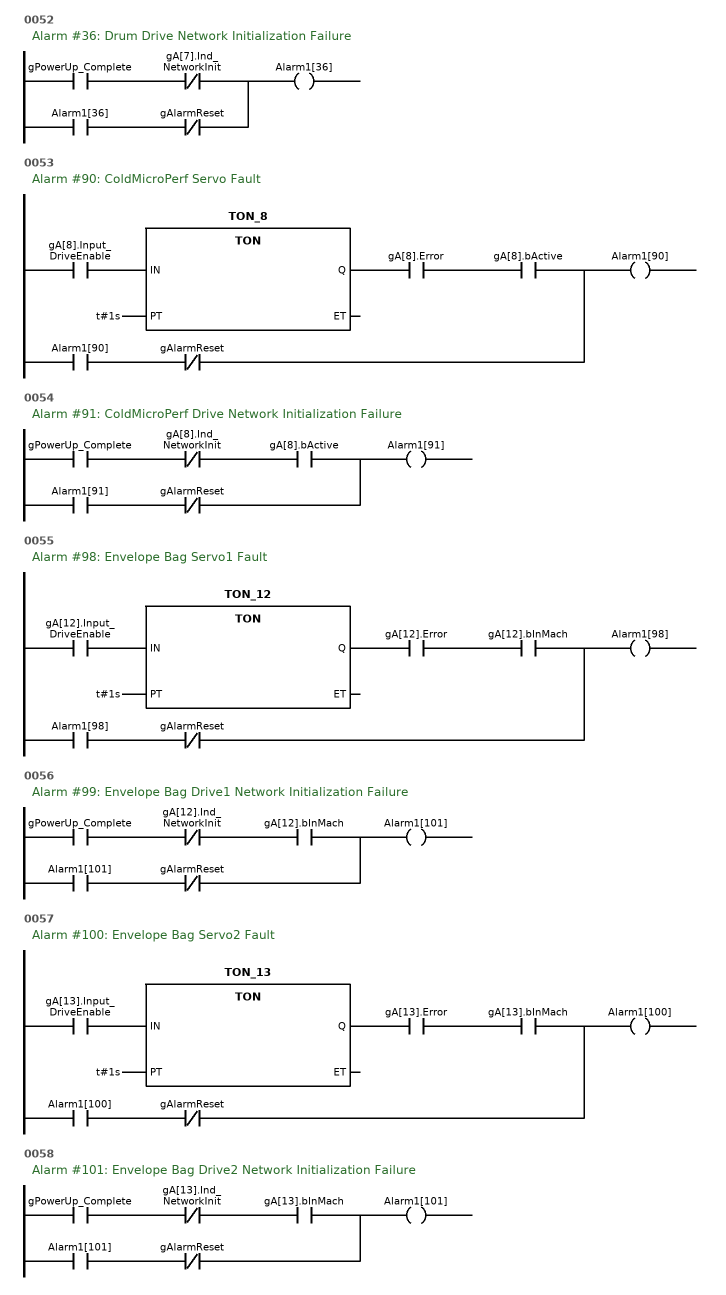
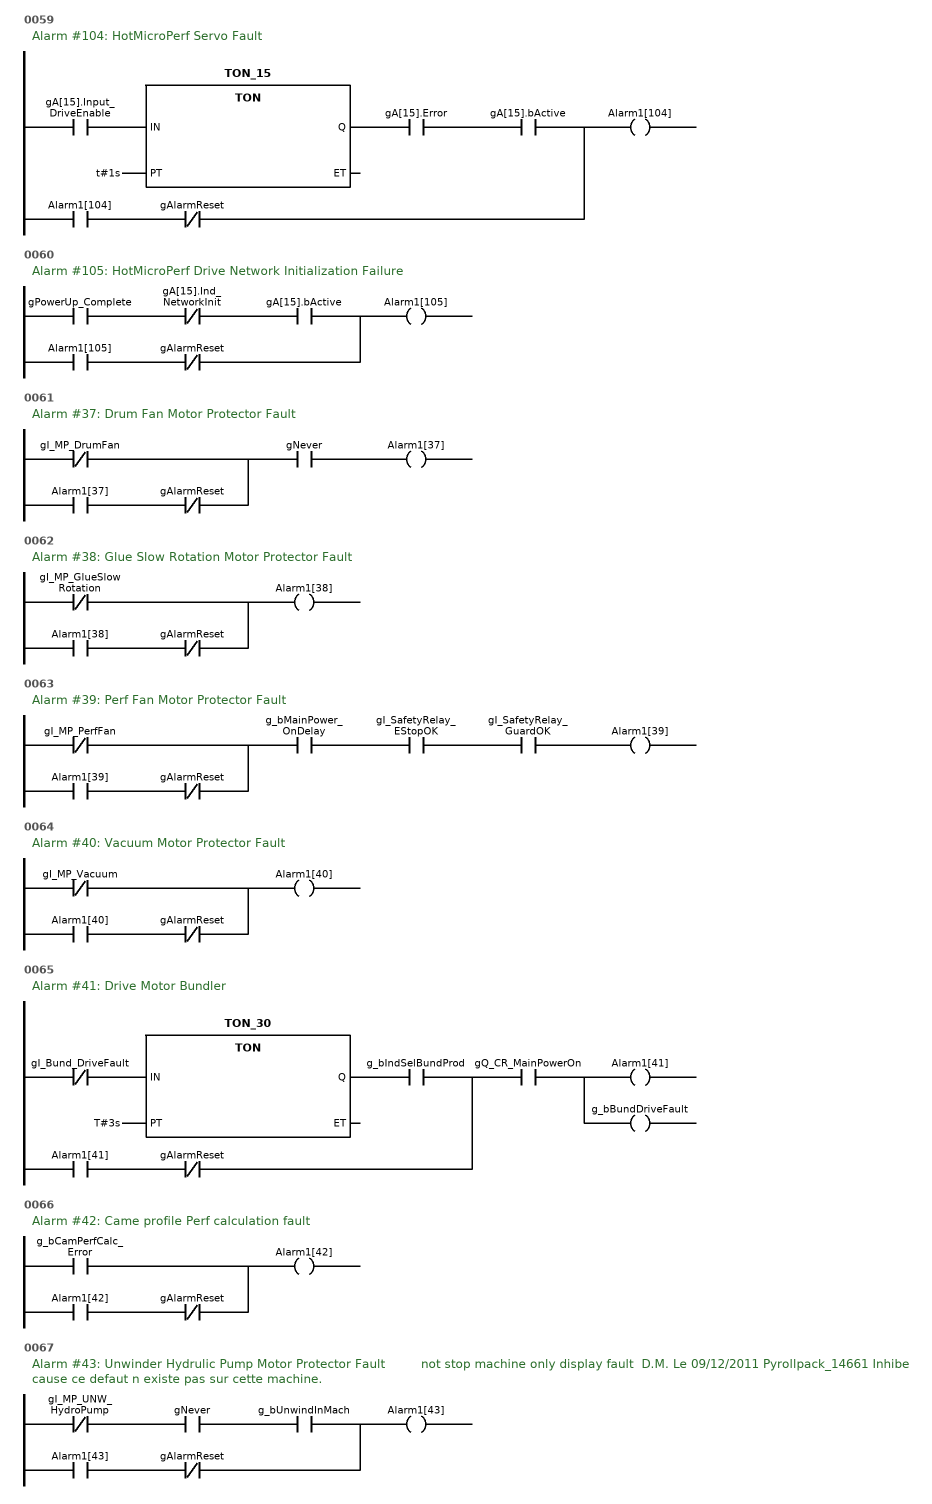
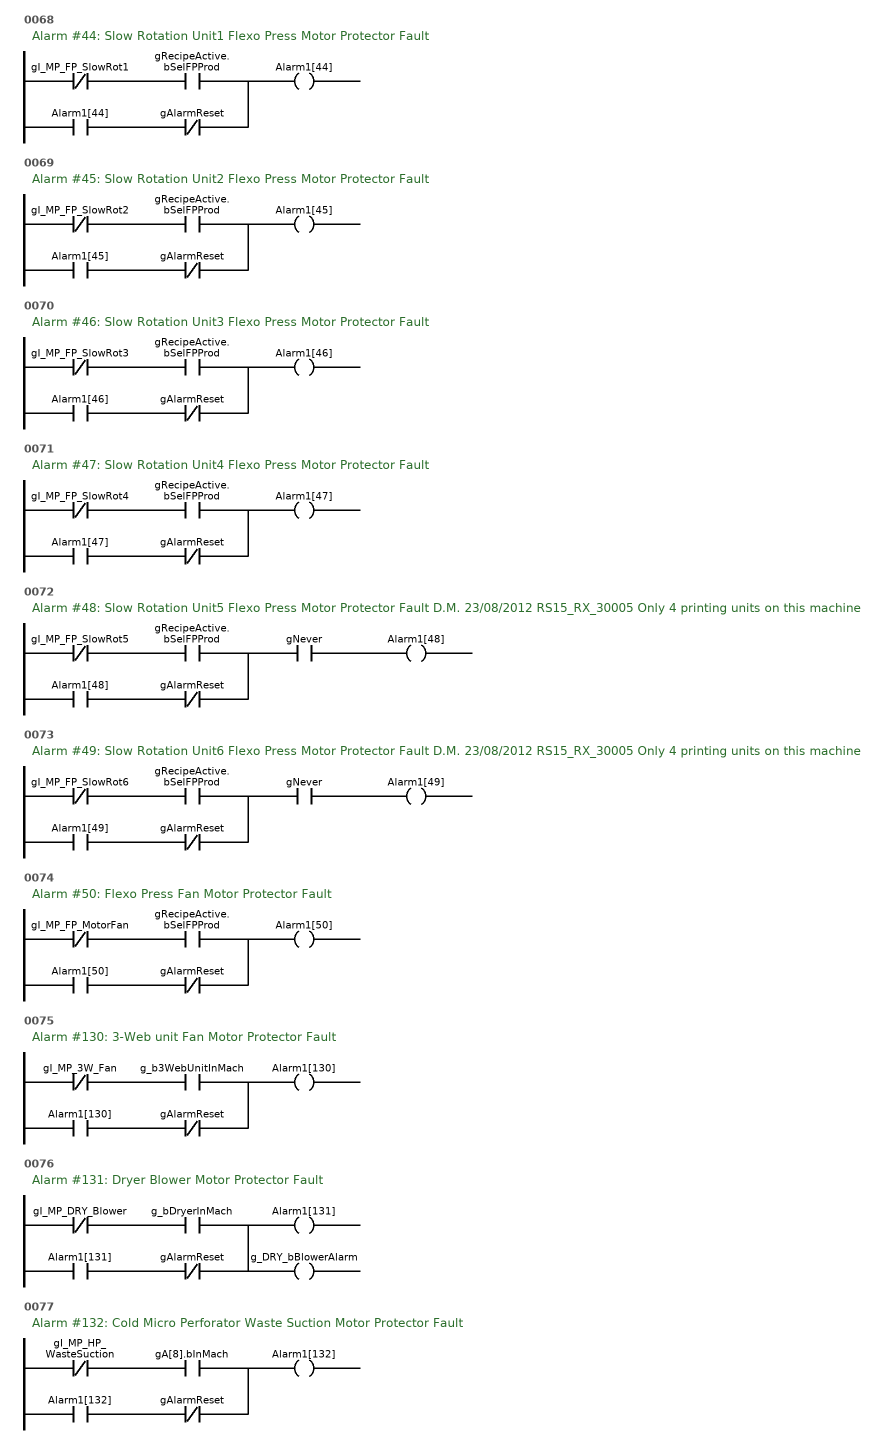
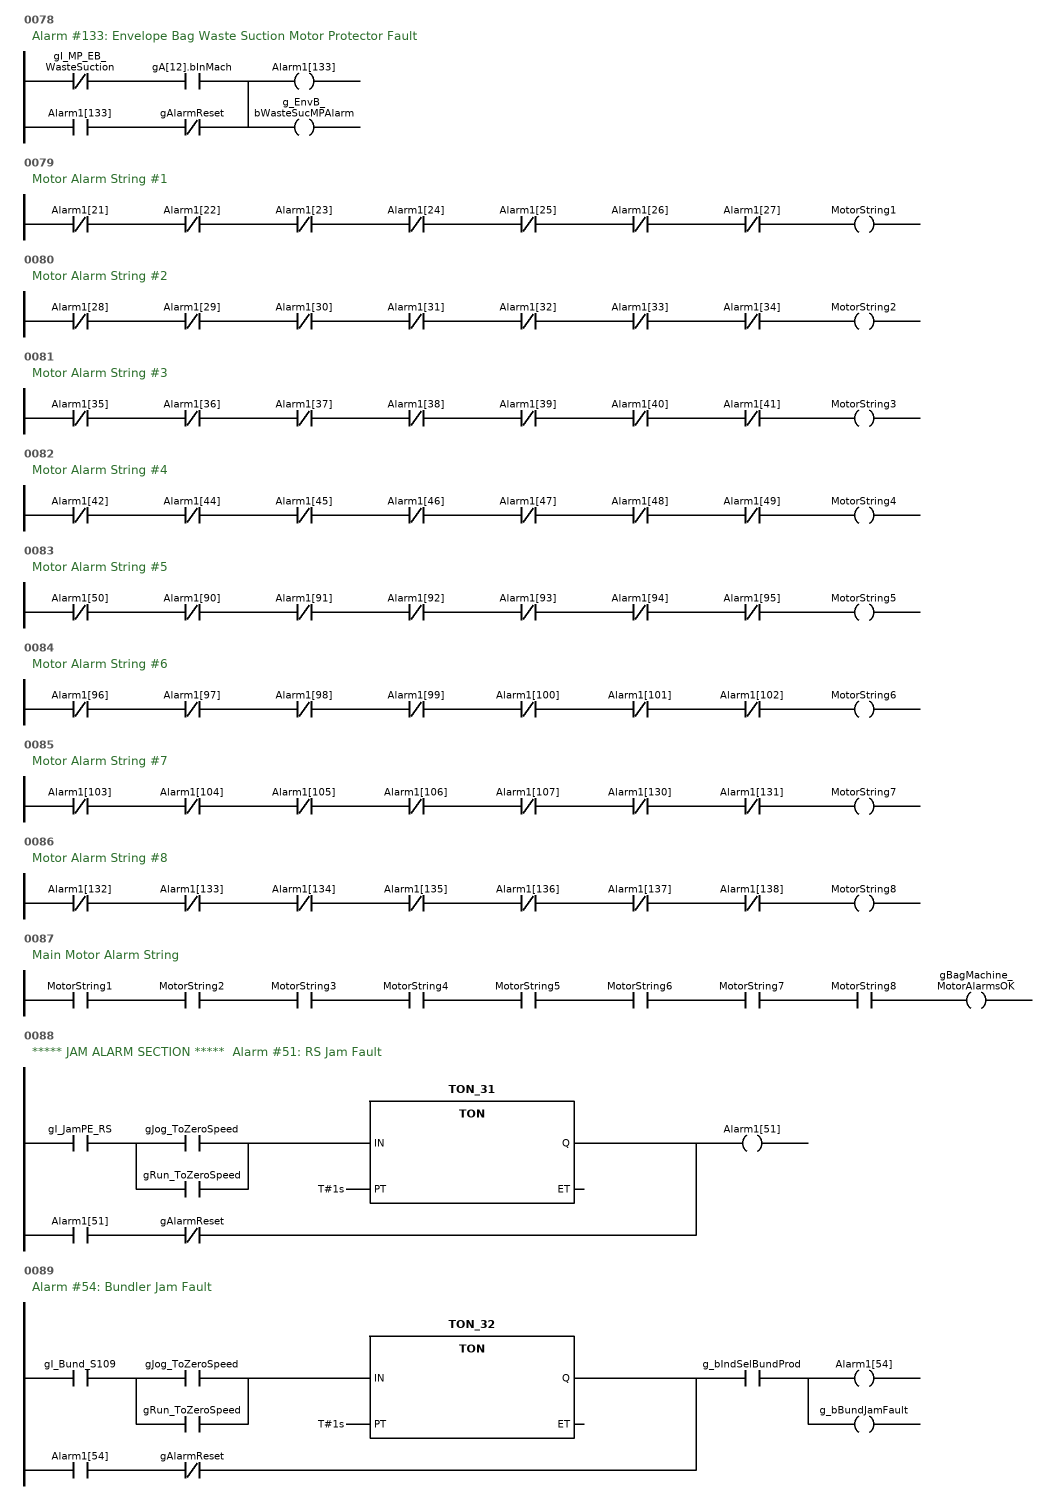
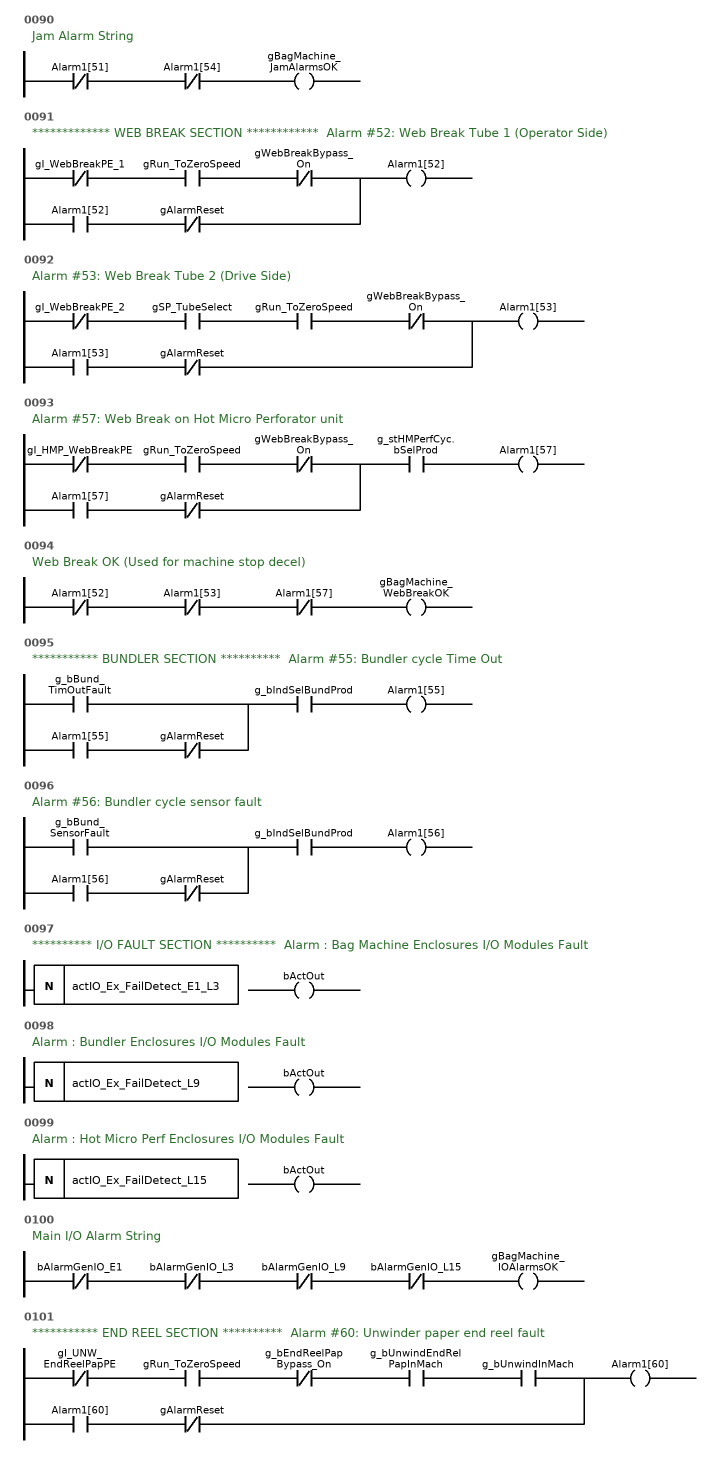
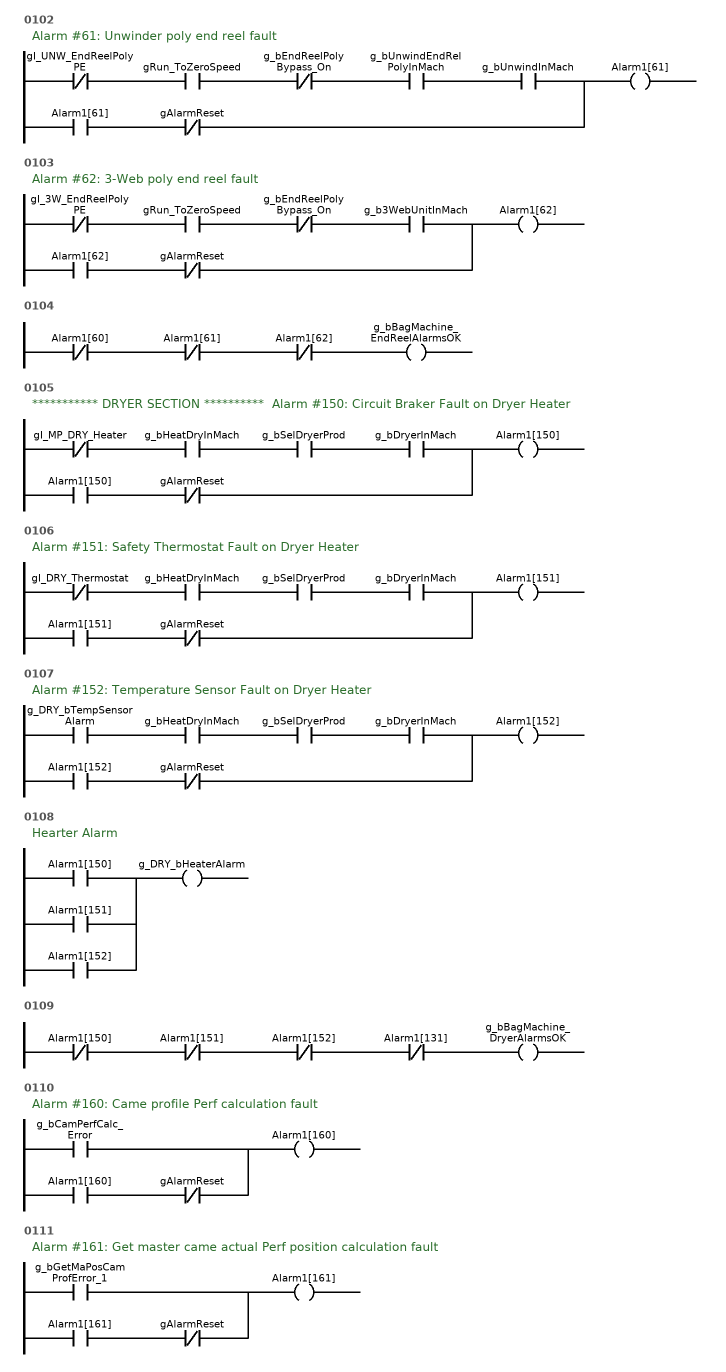
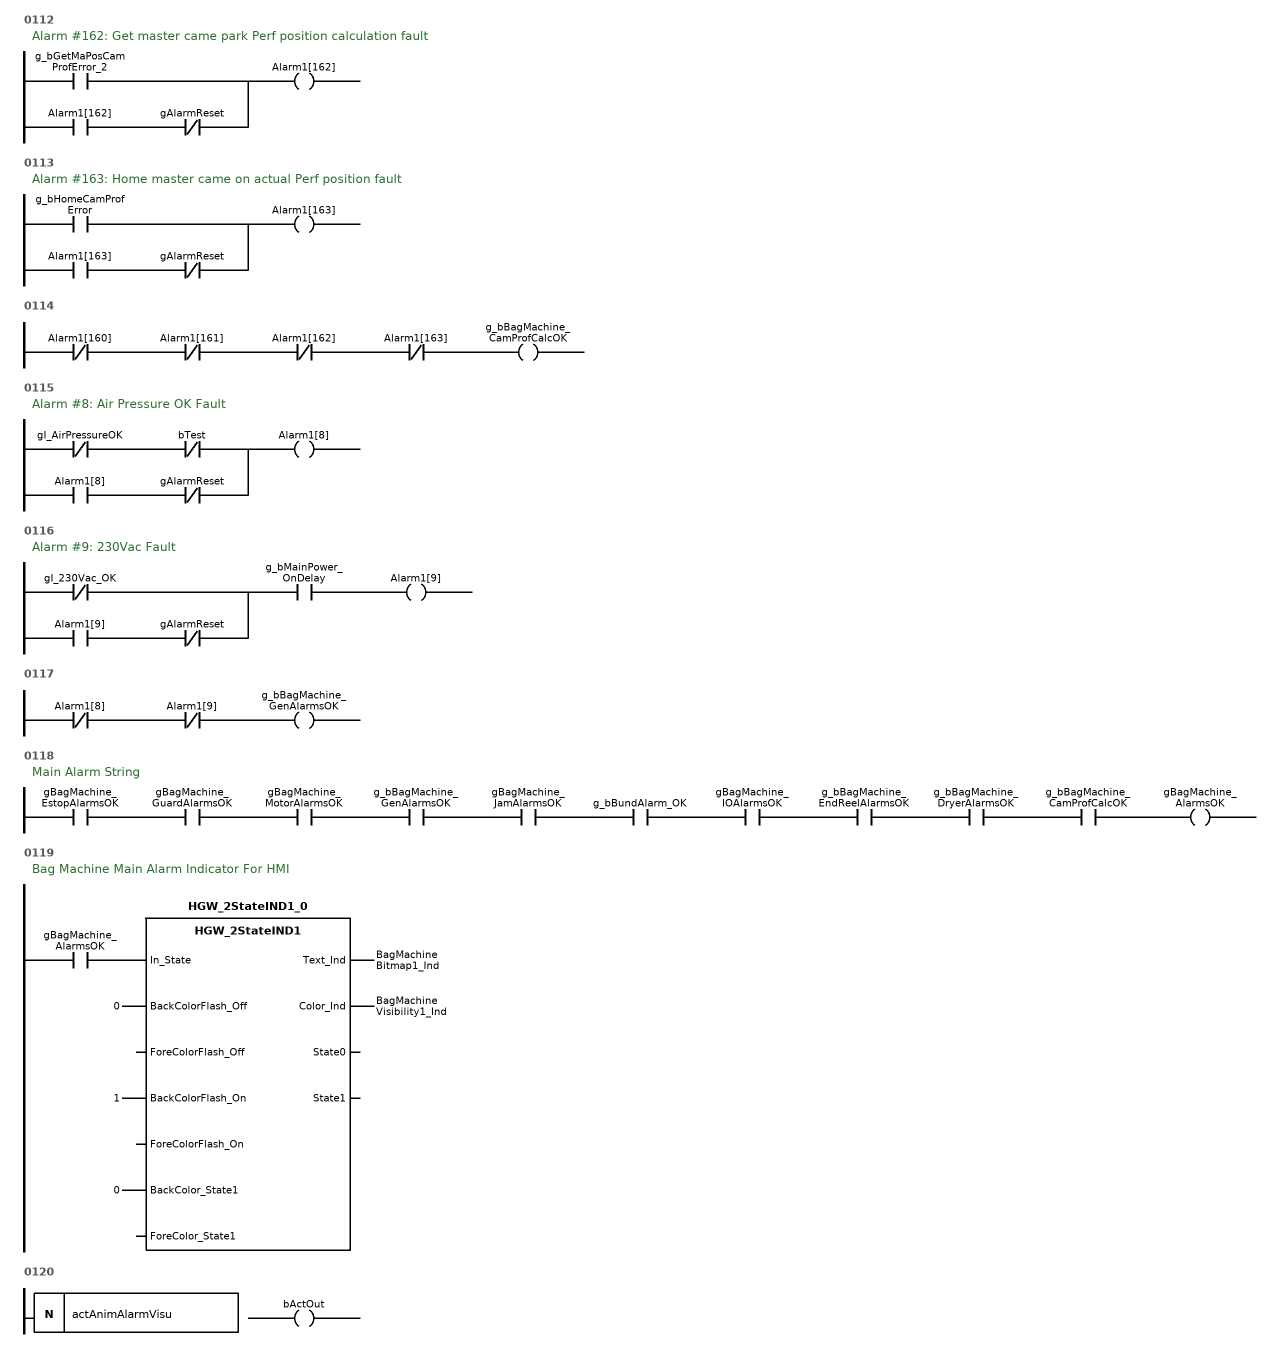
Ladder, written as Structured Text:
```iecst
(********************************************************************
 * COPYRIGHT --
 ********************************************************************
 * Program: Alarms1
 * File: Alarms1Cyclic.ld
 * Author: pkiel
 * Created: September 22, 2009
 ********************************************************************
 * Implementation of program Alarms1
 ********************************************************************)

PROGRAM _CYCLIC
VAR
    _p1 : BOOL;
    _p2 : BOOL;
    _p3 : BOOL;
    _p4 : BOOL;
    _p5 : BOOL;
END_VAR
(* Network 1: ***** E-STOP ALARM SECTION *****  Alarm #1:  E-Stop PB *)
Alarm1[1] := gI_EstopPB_1 OR (Alarm1[1] AND NOT gAlarmReset);

(* Network 2: Alarm #2: Unwind E-Stop PB *)
Alarm1[2] := gI_EstopPB_Unwind OR (Alarm1[2] AND NOT gAlarmReset);

(* Network 3: Alarm #3: E-Stop PB *)
Alarm1[3] := gI_EstopPB_2 OR (Alarm1[3] AND NOT gAlarmReset);

(* Network 4: Alarm #4: E-Stop PB *)
Alarm1[4] := gI_EstopPB_3 OR (Alarm1[4] AND NOT gAlarmReset);

(* Network 5: Alarm #5: E-Stop PB *)
Alarm1[5] := gI_EstopPB_4 OR (Alarm1[5] AND NOT gAlarmReset);

(* Network 6: Alarm #6: E-Stop PB *)
Alarm1[6] := gI_EstopPB_5 OR (Alarm1[6] AND NOT gAlarmReset);

(* Network 7: Alarm #7: Safety E-Stop Relay Fault *)
_p1 := Alarm1[7] AND NOT gAlarmReset;
Alarm1[7] := NOT gI_SafetyRelay_EStopOK OR (Alarm1[7] AND NOT gAlarmReset);
g_bIndEStop := NOT gI_SafetyRelay_EStopOK OR _p1;

(* Network 8: Alarm #20: E-Stop on FootSwitch Jog *)
Alarm1[20] := (gI_JogPB_1 AND NOT gI_SafetyRelay_EStopOK) OR (Alarm1[20] AND NOT gAlarmReset);

(* Network 9: Alarm #10: EStop PB Bundler  *)
Alarm1[10] := gI_Bund_EStopPB OR (Alarm1[10] AND NOT gAlarmReset);

(* Network 10 *)
g_bIndEStopStandstill := (NOT gI_SafetyRelay_EStopOK AND NOT gA[9].Ind_InMotion) OR (g_bIndEStopStandstill AND NOT gAlarmReset AND NOT gA[1].Ind_Enabled AND NOT gA[11].Ind_Enabled AND NOT gA[2].Ind_Enabled AND NOT gA[3].Ind_Enabled AND NOT gA[4].Ind_Enabled AND NOT gA[5].Ind_Enabled AND NOT gA[6].Ind_Enabled AND NOT gA[7].Ind_Enabled AND NOT gA[8].Ind_Enabled AND NOT gA[12].Ind_Enabled AND NOT gA[13].Ind_Enabled AND NOT gA[15].Ind_Enabled);

(* Network 11: Alarm #80: EStop PB on Flexo Press *)
Alarm1[80] := Alarm1[80] AND NOT gAlarmReset;

(* Network 12: Alarm #81: EStop PB on 3-Web Unit *)
Alarm1[81] := (gI_3W_EStopPB AND g_b3WebUnitInMach) OR (Alarm1[81] AND NOT gAlarmReset);

(* Network 13: Alarm #82: EStop PB on Hot Micro Perf *)
Alarm1[82] := gI_HMP_EStopPB OR (Alarm1[82] AND NOT gAlarmReset);

(* Network 14: E-Stop Alarm String 1 *)
EstopString1 := NOT Alarm1[1] AND NOT Alarm1[2] AND NOT Alarm1[3] AND NOT Alarm1[4] AND NOT Alarm1[5] AND NOT Alarm1[6] AND NOT Alarm1[7];

(* Network 15: Main E-Stop Alarm String *)
EstopString2 := EstopString1 AND NOT Alarm1[10] AND NOT g_bIndEStop AND NOT Alarm1[80] AND NOT Alarm1[81];

(* Network 16: Main E-Stop Alarm String *)
gBagMachine_EstopAlarmsOK := EstopString2 AND NOT Alarm1[82] AND NOT Alarm1[83] AND NOT Alarm1[84] AND NOT Alarm1[85] AND NOT Alarm1[86] AND NOT Alarm1[87];

(* Network 17: ***** GUARD ALARM SECTION *****  Guard Alarm Enable Run *)
GuardAlarmEnable := gRun_ToZeroSpeed OR NOT gNever;

(* Network 18: Guard Alarm Enable Jog *)
GuardAlarmEnable1 := gJog_ToZeroSpeed OR NOT gNever;

(* Network 19: Alarm #11: Guard Open *)
Alarm1[11] := (gI_GSW_Door1 AND (GuardAlarmEnable OR GuardAlarmEnable1)) OR (Alarm1[11] AND NOT gAlarmReset);

(* Network 20: Alarm #12: Guard Open *)
Alarm1[12] := (gI_GSW_Door2 AND (GuardAlarmEnable OR GuardAlarmEnable1)) OR (Alarm1[12] AND NOT gAlarmReset);

(* Network 21: Alarm #13: Drum Guard Open *)
Alarm1[13] := (gI_GSW_Drum AND GuardAlarmEnable AND NOT gSetupMode_On) OR (Alarm1[13] AND NOT gAlarmReset);

(* Network 22: Alarm #14: Perf Doors Guard Open *)
Alarm1[14] := ((gI_GSW_PerfDoors OR gI_GSW_PerfDoor2) AND GuardAlarmEnable AND NOT gSetupMode_On) OR (Alarm1[14] AND NOT gAlarmReset);

(* Network 23: Alarm #15: Slitting Door Guard Open *)
Alarm1[15] := (gI_GSW_SlittingDoor AND GuardAlarmEnable AND NOT gSetupMode_On) OR (Alarm1[15] AND NOT gAlarmReset);

(* Network 24: Alarm #16: RS Entry Guard Open *)
Alarm1[16] := (gI_GSW_RSEntry AND (GuardAlarmEnable OR GuardAlarmEnable1)) OR (Alarm1[16] AND NOT gAlarmReset);

(* Network 25: Alarm #17: Tearing Guard Open *)
Alarm1[17] := (gI_GSW_Tearing AND GuardAlarmEnable AND NOT gSetupMode_On) OR (Alarm1[17] AND NOT gAlarmReset);

(* Network 26: Alarm #18: Guard Safety Relay Fault *)
Alarm1[18] := (NOT gI_SafetyRelay_GuardOK AND (GuardAlarmEnable OR GuardAlarmEnable1)) OR (Alarm1[18] AND NOT gAlarmReset);

(* Network 27: Alarm #19: Bundler Guard Open *)
Alarm1[19] := (NOT g_bBundGuard_OK AND (GuardAlarmEnable OR GuardAlarmEnable1) AND g_bIndSelBundProd) OR (Alarm1[19] AND NOT gAlarmReset);

(* Network 28: Alarm #70: Flexo Press Doors Open *)
Alarm1[70] := (gI_GSW_FP_Doors AND (GuardAlarmEnable OR GuardAlarmEnable1) AND gA[2].bInMach) OR (Alarm1[70] AND NOT gAlarmReset);

(* Network 29: Alarm #71: Flexo Press Gates Open *)
Alarm1[71] := (gI_GSW_FP_Gates AND (GuardAlarmEnable OR GuardAlarmEnable1) AND gA[2].bInMach AND NOT gSetupMode_On) OR (Alarm1[71] AND NOT gAlarmReset);

(* Network 30: Guard Flexo *)
g_bFP_GuardFault := Alarm1[70] OR Alarm1[71];

(* Network 31: Alarm #72: 3-Web Unit Guard Open *)
Alarm1[72] := (gI_GSW_3W AND (GuardAlarmEnable OR GuardAlarmEnable1) AND g_b3WebUnitInMach) OR (Alarm1[72] AND NOT gAlarmReset);

(* Network 32: Alarm #73: Hot Micro Perforator Guard Open *)
Alarm1[73] := (gI_GSW_HMPerf AND (GuardAlarmEnable OR GuardAlarmEnable1) AND gA[15].bInMach AND NOT gSetupMode_On) OR (Alarm1[73] AND NOT gAlarmReset);

(* Network 33: Alarm #74: Cold Micro Perforator Gates Open *)
Alarm1[74] := (gI_GSW_CMPerfGates AND (GuardAlarmEnable OR GuardAlarmEnable1) AND gA[8].bInMach AND NOT gSetupMode_On) OR (Alarm1[74] AND NOT gAlarmReset);

(* Network 34: Alarm #75: Cold Micro Perforator Gear Door Open *)
Alarm1[75] := (gI_GSW_CMPerfDoor AND (GuardAlarmEnable OR GuardAlarmEnable1) AND gA[8].bInMach) OR (Alarm1[75] AND NOT gAlarmReset);

(* Network 35: Main Guard Alarm String 1 *)
bGuardString1 := NOT Alarm1[11] AND NOT Alarm1[12] AND NOT Alarm1[13] AND NOT Alarm1[14] AND NOT Alarm1[15] AND NOT Alarm1[16] AND NOT Alarm1[17] AND NOT Alarm1[18] AND NOT Alarm1[19];

(* Network 36: Main Guard Alarm String 2 *)
gBagMachine_GuardAlarmsOK := (bGuardString1 AND NOT Alarm1[70] AND NOT Alarm1[71] AND NOT Alarm1[72] AND NOT Alarm1[73] AND NOT Alarm1[74] AND NOT Alarm1[75] AND NOT Alarm1[76] AND NOT Alarm1[77]) OR g_bBypassGuard;

(* Network 37: *****MOTOR ALARM SECTION *****  Alarm #21: Servo Power Supply Fault *)
Alarm1[21] := gA[0].Error OR (Alarm1[21] AND NOT gAlarmReset);

(* Network 38: Alarm #22: Servo Drive Power Supply Network Initialization Failure *)
Alarm1[22] := (gPowerUp_Complete AND NOT gA[0].Ind_NetworkInit) OR (Alarm1[22] AND NOT gAlarmReset);

(* Network 39: Alarm #23: Perf Servo Fault *)
TON_1(IN := gA[1].Input_DriveEnable, PT := t#1s);
Alarm1[23] := (TON_1.Q AND gA[1].Error) OR (Alarm1[23] AND NOT gAlarmReset);

(* Network 40: Alarm #24: Perf Drive Network Initialization Failure *)
Alarm1[24] := (gPowerUp_Complete AND NOT gA[1].Ind_NetworkInit) OR (Alarm1[24] AND NOT gAlarmReset);

(* Network 41: Alarm #25: Printer Servo Fault *)
TON_2(IN := gA[2].Input_DriveEnable, PT := t#1s);
Alarm1[25] := (TON_2.Q AND gA[2].Error) OR (Alarm1[25] AND NOT gAlarmReset);

(* Network 42: Alarm #26: Printer Drive Network Initialization Failure *)
Alarm1[26] := ((gPowerUp_Complete AND NOT gA[2].Ind_NetworkInit) OR (Alarm1[26] AND NOT gAlarmReset)) AND gNever;

(* Network 43: Alarm #27: Holding (Maintaining) Servo Fault *)
TON_3(IN := gA[3].Input_DriveEnable, PT := t#1s);
Alarm1[27] := (TON_3.Q AND gA[3].Error) OR (Alarm1[27] AND NOT gAlarmReset);

(* Network 44: Alarm #28: Holding (Maintaining) Drive Network Initialization Failure *)
Alarm1[28] := (gPowerUp_Complete AND NOT gA[3].Ind_NetworkInit) OR (Alarm1[28] AND NOT gAlarmReset);

(* Network 45: Alarm #29: Tearing Servo Fault *)
TON_4(IN := gA[4].Input_DriveEnable, PT := t#1s);
Alarm1[29] := (TON_4.Q AND gA[4].Error) OR (Alarm1[29] AND NOT gAlarmReset);

(* Network 46: Alarm #30: TearingDrive Network Initialization Failure *)
Alarm1[30] := (gPowerUp_Complete AND NOT gA[4].Ind_NetworkInit) OR (Alarm1[30] AND NOT gAlarmReset);

(* Network 47: Alarm #31: Entry Pull Roll Servo Fault *)
TON_5(IN := gA[5].Input_DriveEnable, PT := t#1s);
Alarm1[31] := (TON_5.Q AND gA[5].Error) OR (Alarm1[31] AND NOT gAlarmReset);

(* Network 48: Alarm #32: Entry Pull Roll Drive Network Initialization Failure *)
Alarm1[32] := (gPowerUp_Complete AND NOT gA[5].Ind_NetworkInit) OR (Alarm1[32] AND NOT gAlarmReset);

(* Network 49: Alarm #33: Exit Pull Roll Servo Fault *)
TON_6(IN := gA[6].Input_DriveEnable, PT := t#1s);
Alarm1[33] := (TON_6.Q AND gA[6].Error) OR (Alarm1[33] AND NOT gAlarmReset);

(* Network 50: Alarm #34: Exit Pull Roll Drive Network Initialization Failure *)
Alarm1[34] := (gPowerUp_Complete AND NOT gA[6].Ind_NetworkInit) OR (Alarm1[34] AND NOT gAlarmReset);

(* Network 51: Alarm #35: Drum Servo Fault *)
TON_7(IN := gA[7].Input_DriveEnable, PT := t#1s);
Alarm1[35] := (TON_7.Q AND gA[7].Error) OR (Alarm1[35] AND NOT gAlarmReset);

(* Network 52: Alarm #36: Drum Drive Network Initialization Failure *)
Alarm1[36] := (gPowerUp_Complete AND NOT gA[7].Ind_NetworkInit) OR (Alarm1[36] AND NOT gAlarmReset);

(* Network 53: Alarm #90: ColdMicroPerf Servo Fault *)
TON_8(IN := gA[8].Input_DriveEnable, PT := t#1s);
Alarm1[90] := (TON_8.Q AND gA[8].Error AND gA[8].bActive) OR (Alarm1[90] AND NOT gAlarmReset);

(* Network 54: Alarm #91: ColdMicroPerf Drive Network Initialization Failure *)
Alarm1[91] := (gPowerUp_Complete AND NOT gA[8].Ind_NetworkInit AND gA[8].bActive) OR (Alarm1[91] AND NOT gAlarmReset);

(* Network 55: Alarm #98: Envelope Bag Servo1 Fault *)
TON_12(IN := gA[12].Input_DriveEnable, PT := t#1s);
Alarm1[98] := (TON_12.Q AND gA[12].Error AND gA[12].bInMach) OR (Alarm1[98] AND NOT gAlarmReset);

(* Network 56: Alarm #99: Envelope Bag Drive1 Network Initialization Failure *)
Alarm1[101] := (gPowerUp_Complete AND NOT gA[12].Ind_NetworkInit AND gA[12].bInMach) OR (Alarm1[101] AND NOT gAlarmReset);

(* Network 57: Alarm #100: Envelope Bag Servo2 Fault *)
TON_13(IN := gA[13].Input_DriveEnable, PT := t#1s);
Alarm1[100] := (TON_13.Q AND gA[13].Error AND gA[13].bInMach) OR (Alarm1[100] AND NOT gAlarmReset);

(* Network 58: Alarm #101: Envelope Bag Drive2 Network Initialization Failure *)
Alarm1[101] := (gPowerUp_Complete AND NOT gA[13].Ind_NetworkInit AND gA[13].bInMach) OR (Alarm1[101] AND NOT gAlarmReset);

(* Network 59: Alarm #104: HotMicroPerf Servo Fault *)
TON_15(IN := gA[15].Input_DriveEnable, PT := t#1s);
Alarm1[104] := (TON_15.Q AND gA[15].Error AND gA[15].bActive) OR (Alarm1[104] AND NOT gAlarmReset);

(* Network 60: Alarm #105: HotMicroPerf Drive Network Initialization Failure *)
Alarm1[105] := (gPowerUp_Complete AND NOT gA[15].Ind_NetworkInit AND gA[15].bActive) OR (Alarm1[105] AND NOT gAlarmReset);

(* Network 61: Alarm #37: Drum Fan Motor Protector Fault *)
Alarm1[37] := (NOT gI_MP_DrumFan OR (Alarm1[37] AND NOT gAlarmReset)) AND gNever;

(* Network 62: Alarm #38: Glue Slow Rotation Motor Protector Fault *)
Alarm1[38] := NOT gI_MP_GlueSlowRotation OR (Alarm1[38] AND NOT gAlarmReset);

(* Network 63: Alarm #39: Perf Fan Motor Protector Fault *)
Alarm1[39] := (NOT gI_MP_PerfFan OR (Alarm1[39] AND NOT gAlarmReset)) AND g_bMainPower_OnDelay AND gI_SafetyRelay_EStopOK AND gI_SafetyRelay_GuardOK;

(* Network 64: Alarm #40: Vacuum Motor Protector Fault *)
Alarm1[40] := NOT gI_MP_Vacuum OR (Alarm1[40] AND NOT gAlarmReset);

(* Network 65: Alarm #41: Drive Motor Bundler *)
TON_30(IN := NOT gI_Bund_DriveFault, PT := T#3s);
_p2 := ((TON_30.Q AND g_bIndSelBundProd) OR (Alarm1[41] AND NOT gAlarmReset)) AND gQ_CR_MainPowerOn;
Alarm1[41] := _p2;
g_bBundDriveFault := _p2;

(* Network 66: Alarm #42: Came profile Perf calculation fault  *)
Alarm1[42] := g_bCamPerfCalc_Error OR (Alarm1[42] AND NOT gAlarmReset);

(* Network 67: Alarm #43: Unwinder Hydrulic Pump Motor Protector Fault         not stop machine only display fault  D.M. Le 09/12/2011 Pyrollpack_14661 Inhibe cause ce defaut n existe pas sur cette machine. *)
Alarm1[43] := (NOT gI_MP_UNW_HydroPump AND gNever AND g_bUnwindInMach) OR (Alarm1[43] AND NOT gAlarmReset);

(* Network 68: Alarm #44: Slow Rotation Unit1 Flexo Press Motor Protector Fault *)
Alarm1[44] := (NOT gI_MP_FP_SlowRot1 AND gRecipeActive.bSelFPProd) OR (Alarm1[44] AND NOT gAlarmReset);

(* Network 69: Alarm #45: Slow Rotation Unit2 Flexo Press Motor Protector Fault *)
Alarm1[45] := (NOT gI_MP_FP_SlowRot2 AND gRecipeActive.bSelFPProd) OR (Alarm1[45] AND NOT gAlarmReset);

(* Network 70: Alarm #46: Slow Rotation Unit3 Flexo Press Motor Protector Fault *)
Alarm1[46] := (NOT gI_MP_FP_SlowRot3 AND gRecipeActive.bSelFPProd) OR (Alarm1[46] AND NOT gAlarmReset);

(* Network 71: Alarm #47: Slow Rotation Unit4 Flexo Press Motor Protector Fault *)
Alarm1[47] := (NOT gI_MP_FP_SlowRot4 AND gRecipeActive.bSelFPProd) OR (Alarm1[47] AND NOT gAlarmReset);

(* Network 72: Alarm #48: Slow Rotation Unit5 Flexo Press Motor Protector Fault D.M. 23/08/2012 RS15_RX_30005 Only 4 printing units on this machine  *)
Alarm1[48] := ((NOT gI_MP_FP_SlowRot5 AND gRecipeActive.bSelFPProd) OR (Alarm1[48] AND NOT gAlarmReset)) AND gNever;

(* Network 73: Alarm #49: Slow Rotation Unit6 Flexo Press Motor Protector Fault D.M. 23/08/2012 RS15_RX_30005 Only 4 printing units on this machine  *)
Alarm1[49] := ((NOT gI_MP_FP_SlowRot6 AND gRecipeActive.bSelFPProd) OR (Alarm1[49] AND NOT gAlarmReset)) AND gNever;

(* Network 74: Alarm #50: Flexo Press Fan Motor Protector Fault *)
Alarm1[50] := (NOT gI_MP_FP_MotorFan AND gRecipeActive.bSelFPProd) OR (Alarm1[50] AND NOT gAlarmReset);

(* Network 75: Alarm #130: 3-Web unit Fan Motor Protector Fault *)
Alarm1[130] := (NOT gI_MP_3W_Fan AND g_b3WebUnitInMach) OR (Alarm1[130] AND NOT gAlarmReset);

(* Network 76: Alarm #131: Dryer Blower Motor Protector Fault *)
_p3 := Alarm1[131] AND NOT gAlarmReset;
Alarm1[131] := (NOT gI_MP_DRY_Blower AND g_bDryerInMach) OR (Alarm1[131] AND NOT gAlarmReset);
g_DRY_bBlowerAlarm := (NOT gI_MP_DRY_Blower AND g_bDryerInMach) OR _p3;

(* Network 77: Alarm #132: Cold Micro Perforator Waste Suction Motor Protector Fault *)
Alarm1[132] := (NOT gI_MP_HP_WasteSuction AND gA[8].bInMach) OR (Alarm1[132] AND NOT gAlarmReset);

(* Network 78: Alarm #133: Envelope Bag Waste Suction Motor Protector Fault *)
_p4 := Alarm1[133] AND NOT gAlarmReset;
Alarm1[133] := (NOT gI_MP_EB_WasteSuction AND gA[12].bInMach) OR (Alarm1[133] AND NOT gAlarmReset);
g_EnvB_bWasteSucMPAlarm := (NOT gI_MP_EB_WasteSuction AND gA[12].bInMach) OR _p4;

(* Network 79: Motor Alarm String #1 *)
MotorString1 := NOT Alarm1[21] AND NOT Alarm1[22] AND NOT Alarm1[23] AND NOT Alarm1[24] AND NOT Alarm1[25] AND NOT Alarm1[26] AND NOT Alarm1[27];

(* Network 80: Motor Alarm String #2 *)
MotorString2 := NOT Alarm1[28] AND NOT Alarm1[29] AND NOT Alarm1[30] AND NOT Alarm1[31] AND NOT Alarm1[32] AND NOT Alarm1[33] AND NOT Alarm1[34];

(* Network 81: Motor Alarm String #3 *)
MotorString3 := NOT Alarm1[35] AND NOT Alarm1[36] AND NOT Alarm1[37] AND NOT Alarm1[38] AND NOT Alarm1[39] AND NOT Alarm1[40] AND NOT Alarm1[41];

(* Network 82: Motor Alarm String #4 *)
MotorString4 := NOT Alarm1[42] AND NOT Alarm1[44] AND NOT Alarm1[45] AND NOT Alarm1[46] AND NOT Alarm1[47] AND NOT Alarm1[48] AND NOT Alarm1[49];

(* Network 83: Motor Alarm String #5 *)
MotorString5 := NOT Alarm1[50] AND NOT Alarm1[90] AND NOT Alarm1[91] AND NOT Alarm1[92] AND NOT Alarm1[93] AND NOT Alarm1[94] AND NOT Alarm1[95];

(* Network 84: Motor Alarm String #6 *)
MotorString6 := NOT Alarm1[96] AND NOT Alarm1[97] AND NOT Alarm1[98] AND NOT Alarm1[99] AND NOT Alarm1[100] AND NOT Alarm1[101] AND NOT Alarm1[102];

(* Network 85: Motor Alarm String #7 *)
MotorString7 := NOT Alarm1[103] AND NOT Alarm1[104] AND NOT Alarm1[105] AND NOT Alarm1[106] AND NOT Alarm1[107] AND NOT Alarm1[130] AND NOT Alarm1[131];

(* Network 86: Motor Alarm String #8 *)
MotorString8 := NOT Alarm1[132] AND NOT Alarm1[133] AND NOT Alarm1[134] AND NOT Alarm1[135] AND NOT Alarm1[136] AND NOT Alarm1[137] AND NOT Alarm1[138];

(* Network 87: Main Motor Alarm String *)
gBagMachine_MotorAlarmsOK := MotorString1 AND MotorString2 AND MotorString3 AND MotorString4 AND MotorString5 AND MotorString6 AND MotorString7 AND MotorString8;

(* Network 88: ***** JAM ALARM SECTION *****  Alarm #51: RS Jam Fault *)
TON_31(IN := gI_JamPE_RS AND (gJog_ToZeroSpeed OR gRun_ToZeroSpeed), PT := T#1s);
Alarm1[51] := (Alarm1[51] AND NOT gAlarmReset) OR TON_31.Q;

(* Network 89: Alarm #54: Bundler Jam Fault *)
TON_32(IN := gI_Bund_S109 AND (gJog_ToZeroSpeed OR gRun_ToZeroSpeed), PT := T#1s);
_p5 := ((Alarm1[54] AND NOT gAlarmReset) OR TON_32.Q) AND g_bIndSelBundProd;
Alarm1[54] := _p5;
g_bBundJamFault := _p5;

(* Network 90: Jam Alarm String *)
gBagMachine_JamAlarmsOK := NOT Alarm1[51] AND NOT Alarm1[54];

(* Network 91: ************* WEB BREAK SECTION ************  Alarm #52: Web Break Tube 1 (Operator Side) *)
Alarm1[52] := (NOT gI_WebBreakPE_1 AND gRun_ToZeroSpeed AND NOT gWebBreakBypass_On) OR (Alarm1[52] AND NOT gAlarmReset);

(* Network 92: Alarm #53: Web Break Tube 2 (Drive Side) *)
Alarm1[53] := (NOT gI_WebBreakPE_2 AND gSP_TubeSelect AND gRun_ToZeroSpeed AND NOT gWebBreakBypass_On) OR (Alarm1[53] AND NOT gAlarmReset);

(* Network 93: Alarm #57: Web Break on Hot Micro Perforator unit  *)
Alarm1[57] := ((NOT gI_HMP_WebBreakPE AND gRun_ToZeroSpeed AND NOT gWebBreakBypass_On) OR (Alarm1[57] AND NOT gAlarmReset)) AND g_stHMPerfCyc.bSelProd;

(* Network 94: Web Break OK (Used for machine stop decel) *)
gBagMachine_WebBreakOK := NOT Alarm1[52] AND NOT Alarm1[53] AND NOT Alarm1[57];

(* Network 95: *********** BUNDLER SECTION **********  Alarm #55: Bundler cycle Time Out *)
Alarm1[55] := (g_bBund_TimOutFault OR (Alarm1[55] AND NOT gAlarmReset)) AND g_bIndSelBundProd;

(* Network 96: Alarm #56: Bundler cycle sensor fault *)
Alarm1[56] := (g_bBund_SensorFault OR (Alarm1[56] AND NOT gAlarmReset)) AND g_bIndSelBundProd;

(* Network 97: ********** I/O FAULT SECTION **********  Alarm : Bag Machine Enclosures I/O Modules Fault  *)
actIO_Ex_FailDetect_E1_L3;
bActOut := FALSE;

(* Network 98: Alarm : Bundler Enclosures I/O Modules Fault  *)
actIO_Ex_FailDetect_L9;
bActOut := FALSE;

(* Network 99: Alarm : Hot Micro Perf Enclosures I/O Modules Fault  *)
actIO_Ex_FailDetect_L15;
bActOut := FALSE;

(* Network 100: Main I/O Alarm String *)
gBagMachine_IOAlarmsOK := NOT bAlarmGenIO_E1 AND NOT bAlarmGenIO_L3 AND NOT bAlarmGenIO_L9 AND NOT bAlarmGenIO_L15;

(* Network 101: *********** END REEL SECTION **********  Alarm #60: Unwinder paper end reel fault *)
Alarm1[60] := (NOT gI_UNW_EndReelPapPE AND gRun_ToZeroSpeed AND NOT g_bEndReelPapBypass_On AND g_bUnwindEndRelPapInMach AND g_bUnwindInMach) OR (Alarm1[60] AND NOT gAlarmReset);

(* Network 102: Alarm #61: Unwinder poly end reel fault *)
Alarm1[61] := (NOT gI_UNW_EndReelPolyPE AND gRun_ToZeroSpeed AND NOT g_bEndReelPolyBypass_On AND g_bUnwindEndRelPolyInMach AND g_bUnwindInMach) OR (Alarm1[61] AND NOT gAlarmReset);

(* Network 103: Alarm #62: 3-Web poly end reel fault *)
Alarm1[62] := (NOT gI_3W_EndReelPolyPE AND gRun_ToZeroSpeed AND NOT g_bEndReelPolyBypass_On AND g_b3WebUnitInMach) OR (Alarm1[62] AND NOT gAlarmReset);

(* Network 104 *)
g_bBagMachine_EndReelAlarmsOK := NOT Alarm1[60] AND NOT Alarm1[61] AND NOT Alarm1[62];

(* Network 105: *********** DRYER SECTION **********  Alarm #150: Circuit Braker Fault on Dryer Heater *)
Alarm1[150] := (NOT gI_MP_DRY_Heater AND g_bHeatDryInMach AND g_bSelDryerProd AND g_bDryerInMach) OR (Alarm1[150] AND NOT gAlarmReset);

(* Network 106: Alarm #151: Safety Thermostat Fault on Dryer Heater *)
Alarm1[151] := (NOT gI_DRY_Thermostat AND g_bHeatDryInMach AND g_bSelDryerProd AND g_bDryerInMach) OR (Alarm1[151] AND NOT gAlarmReset);

(* Network 107: Alarm #152: Temperature Sensor Fault on Dryer Heater *)
Alarm1[152] := (g_DRY_bTempSensorAlarm AND g_bHeatDryInMach AND g_bSelDryerProd AND g_bDryerInMach) OR (Alarm1[152] AND NOT gAlarmReset);

(* Network 108: Hearter Alarm *)
g_DRY_bHeaterAlarm := Alarm1[150] OR Alarm1[151] OR Alarm1[152];

(* Network 109 *)
g_bBagMachine_DryerAlarmsOK := NOT Alarm1[150] AND NOT Alarm1[151] AND NOT Alarm1[152] AND NOT Alarm1[131];

(* Network 110: Alarm #160: Came profile Perf calculation fault  *)
Alarm1[160] := g_bCamPerfCalc_Error OR (Alarm1[160] AND NOT gAlarmReset);

(* Network 111: Alarm #161: Get master came actual Perf position calculation fault  *)
Alarm1[161] := g_bGetMaPosCamProfError_1 OR (Alarm1[161] AND NOT gAlarmReset);

(* Network 112: Alarm #162: Get master came park Perf position calculation fault  *)
Alarm1[162] := g_bGetMaPosCamProfError_2 OR (Alarm1[162] AND NOT gAlarmReset);

(* Network 113: Alarm #163: Home master came on actual Perf position fault  *)
Alarm1[163] := g_bHomeCamProfError OR (Alarm1[163] AND NOT gAlarmReset);

(* Network 114 *)
g_bBagMachine_CamProfCalcOK := NOT Alarm1[160] AND NOT Alarm1[161] AND NOT Alarm1[162] AND NOT Alarm1[163];

(* Network 115: Alarm #8: Air Pressure OK Fault *)
Alarm1[8] := (NOT gI_AirPressureOK AND NOT bTest) OR (Alarm1[8] AND NOT gAlarmReset);

(* Network 116: Alarm #9: 230Vac Fault *)
Alarm1[9] := (NOT gI_230Vac_OK OR (Alarm1[9] AND NOT gAlarmReset)) AND g_bMainPower_OnDelay;

(* Network 117 *)
g_bBagMachine_GenAlarmsOK := NOT Alarm1[8] AND NOT Alarm1[9];

(* Network 118: Main Alarm String *)
gBagMachine_AlarmsOK := gBagMachine_EstopAlarmsOK AND gBagMachine_GuardAlarmsOK AND gBagMachine_MotorAlarmsOK AND g_bBagMachine_GenAlarmsOK AND gBagMachine_JamAlarmsOK AND g_bBundAlarm_OK AND gBagMachine_IOAlarmsOK AND g_bBagMachine_EndReelAlarmsOK AND g_bBagMachine_DryerAlarmsOK AND g_bBagMachine_CamProfCalcOK;

(* Network 119: Bag Machine Main Alarm Indicator For HMI *)
HGW_2StateIND1_0(In_State := gBagMachine_AlarmsOK, BackColorFlash_Off := 0, BackColorFlash_On := 1, BackColor_State1 := 0);
BagMachineBitmap1_Ind := HGW_2StateIND1_0.Text_Ind;
BagMachineVisibility1_Ind := HGW_2StateIND1_0.Color_Ind;

(* Network 120 *)
actAnimAlarmVisu;
bActOut := FALSE;
END_PROGRAM
```

- Program Logical/SupervisoryControl_Section/Alarm_Section/MainAlarms (IEC) - Main Alarm Monitoring (no source held here)

### Program Logical/SupervisoryControl_Section/Guard_Mon (IEC)

#### Guard_Mon.var - Local variables
```iecst
(********************************************************************
 * COPYRIGHT --
 ********************************************************************
 * Program: Guard_Mon
 * File: Guard_Mon.var
 * Author: pkiel
 * Created: October 13, 2009
 ********************************************************************
 * Local variables of program Guard_Mon
 ********************************************************************)
VAR
	BagMachine_GuardsOK : BOOL;
	HGW_2StateIND_0 : HGW_2StateIND;
	GuardsOKColor_Ind : UINT;
END_VAR
```

### Program Logical/SupervisoryControl_Section/HourMeter (IEC)

#### HourMeter.var - Local variables
```iecst
(********************************************************************
 * COPYRIGHT --
 ********************************************************************
 * Program: HourMeter
 * File: HourMeter.var
 * Author: pkiel
 * Created: December 04, 2009
 ********************************************************************
 * Local variables of program HourMeter
 ********************************************************************)
VAR
	HourMeterDisplay : REAL;
END_VAR
```

### Program Logical/SupervisoryControl_Section/Jog (IEC)

#### JogCyclic.ld - Cyclic code
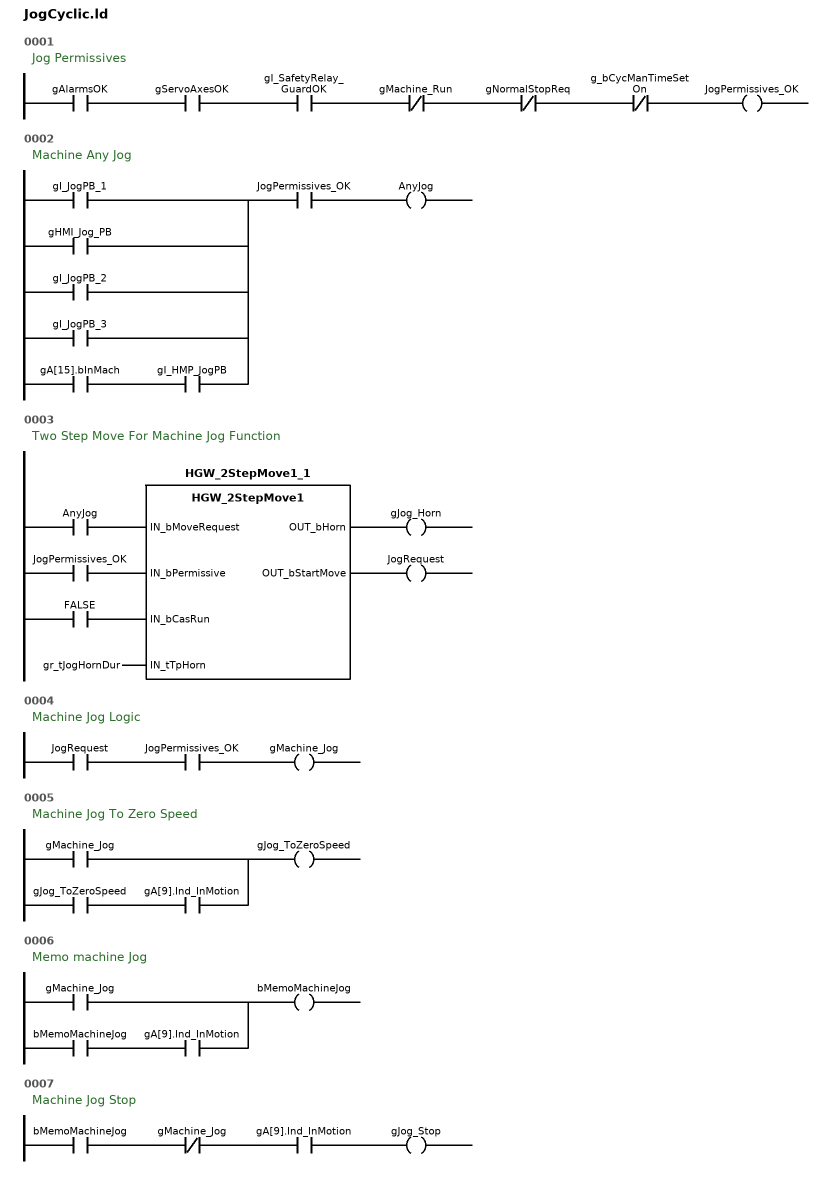
Ladder, written as Structured Text:
```iecst
(********************************************************************
 * COPYRIGHT --
 ********************************************************************
 * Program: Jog
 * File: JogCyclic.ld
 * Author: pkiel
 * Created: October 13, 2009
 ********************************************************************
 * Implementation of program Jog
 ********************************************************************)

PROGRAM _CYCLIC
(* Network 1: Jog Permissives *)
JogPermissives_OK := gAlarmsOK AND gServoAxesOK AND gI_SafetyRelay_GuardOK AND NOT gMachine_Run AND NOT gNormalStopReq AND NOT g_bCycManTimeSetOn;

(* Network 2: Machine Any Jog *)
AnyJog := (gI_JogPB_1 OR gHMI_Jog_PB OR gI_JogPB_2 OR gI_JogPB_3 OR (gA[15].bInMach AND gI_HMP_JogPB)) AND JogPermissives_OK;

(* Network 3: Two Step Move For Machine Jog Function *)
HGW_2StepMove1_1(IN_bMoveRequest := AnyJog, IN_bPermissive := JogPermissives_OK, IN_bCasRun := FALSE, IN_tTpHorn := gr_tJogHornDur);
gJog_Horn := HGW_2StepMove1_1.OUT_bHorn;
JogRequest := HGW_2StepMove1_1.OUT_bStartMove;

(* Network 4: Machine Jog Logic *)
gMachine_Jog := JogRequest AND JogPermissives_OK;

(* Network 5: Machine Jog To Zero Speed *)
gJog_ToZeroSpeed := gMachine_Jog OR (gJog_ToZeroSpeed AND gA[9].Ind_InMotion);

(* Network 6: Memo machine Jog *)
bMemoMachineJog := gMachine_Jog OR (bMemoMachineJog AND gA[9].Ind_InMotion);

(* Network 7: Machine Jog Stop *)
gJog_Stop := bMemoMachineJog AND NOT gMachine_Jog AND gA[9].Ind_InMotion;
END_PROGRAM
```

### Program Logical/SupervisoryControl_Section/ManMode (IEC)

#### ManModeInit.st - Initialization code
```iecst
(********************************************************************
 * COPYRIGHT -- Microsoft
 ********************************************************************
 * Program: ManMode
 * File: ManModeInit.st
 * Author: pkiel
 * Created: July 22, 2011
 ********************************************************************
 * Implementation of program ManMode
 ********************************************************************)

PROGRAM _INIT

(* Manual Mode Off/On PB Colors *)
	HGW_2StatePB_0.BackColor_State0 := gGreen;
	HGW_2StatePB_0.ForeColor_State0 := gBlack;
	HGW_2StatePB_0.BackColor_State1 := gYellow;
	HGW_2StatePB_0.ForeColor_State1 := gBlack;

END_PROGRAM
```

### Program Logical/SupervisoryControl_Section/PowerTimer

#### PowerTimer.var
```iecst
(********************************************************************
 * COPYRIGHT --
 ********************************************************************
 * Program: PowerTimer
 * File: PowerTimer.var
 * Author: pkiel
 * Created: November 04, 2009
 ********************************************************************
 * Local variables of program PowerTimer
 ********************************************************************)
VAR
  TON_0    : TON;
  stTON_1  : TON;
  stPowOff : BOOL ;
  stPowOn  : BOOL ;

  bQ_PL_MainPower : BOOL ;
  bFlash          : BOOL ;
END_VAR
```

#### PowerTimerCyclic.ld
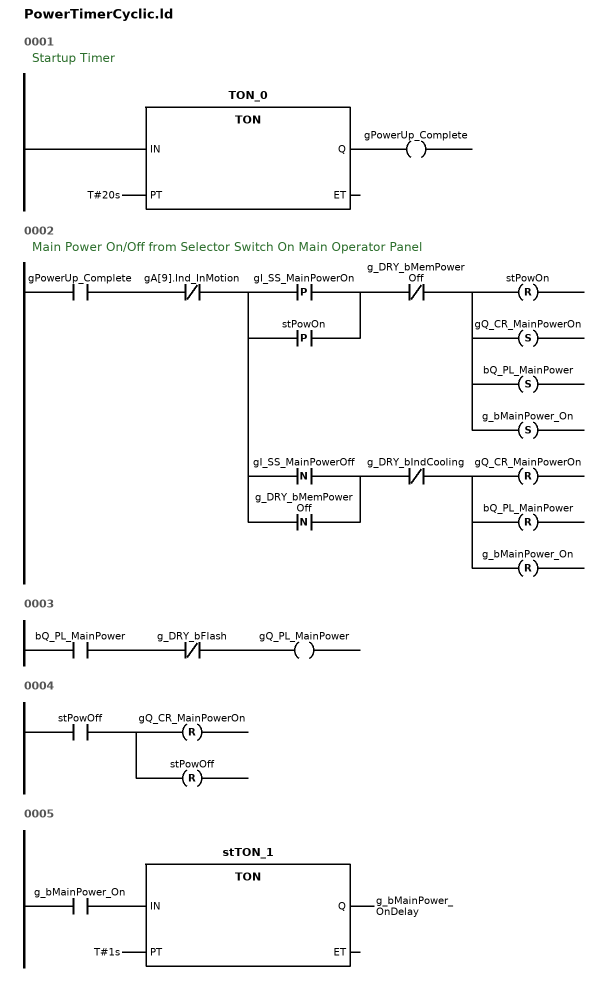
Ladder, written as Structured Text:
```iecst
(********************************************************************
 * COPYRIGHT --
 ********************************************************************
 * Program: PowerTimer
 * File: PowerTimerCyclic.ld
 * Author: pkiel
 * Created: November 04, 2009
 ********************************************************************
 * Implementation of program PowerTimer
 ********************************************************************)

PROGRAM _CYCLIC
VAR
    _e1 : R_TRIG;
    _e2 : R_TRIG;
    _p3 : BOOL;
    _e4 : F_TRIG;
    _e5 : F_TRIG;
    _p6 : BOOL;
END_VAR
(* Network 1: Startup Timer *)
TON_0(IN := TRUE, PT := T#20s);
gPowerUp_Complete := TON_0.Q;

(* Network 2: Main Power On/Off from Selector Switch On Main Operator Panel *)
_e1(CLK := gI_SS_MainPowerOn);
_e2(CLK := stPowOn);
_p3 := gPowerUp_Complete AND NOT gA[9].Ind_InMotion AND (_e1.Q OR _e2.Q) AND NOT g_DRY_bMemPowerOff;
IF _p3 THEN
    stPowOn := FALSE;
    gQ_CR_MainPowerOn := TRUE;
    bQ_PL_MainPower := TRUE;
    g_bMainPower_On := TRUE;
END_IF;
_e4(CLK := gI_SS_MainPowerOff);
_e5(CLK := g_DRY_bMemPowerOff);
_p6 := gPowerUp_Complete AND NOT gA[9].Ind_InMotion AND (_e4.Q OR _e5.Q) AND NOT g_DRY_bIndCooling;
IF _p6 THEN
    gQ_CR_MainPowerOn := FALSE;
    bQ_PL_MainPower := FALSE;
    g_bMainPower_On := FALSE;
END_IF;

(* Network 3 *)
gQ_PL_MainPower := bQ_PL_MainPower AND NOT g_DRY_bFlash;

(* Network 4 *)
IF stPowOff THEN
    gQ_CR_MainPowerOn := FALSE;
    stPowOff := FALSE;
END_IF;

(* Network 5 *)
stTON_1(IN := g_bMainPower_On, PT := T#1s);
g_bMainPower_OnDelay := stTON_1.Q;
END_PROGRAM
```

### Program Logical/SupervisoryControl_Section/Revision (IEC)

#### RevisionCyclic.st - Cyclic code
```iecst
(********************************************************************
 * COPYRIGHT --
 ********************************************************************
 * Program: Revision
 * File: RevisionCyclic.st
 * Author: pkiel
 * Created: December 14, 2009
 ********************************************************************
 * Implementation of program Revision
 ********************************************************************)

PROGRAM _CYCLIC

	CurrentSoftwareRevision := 1.1;

END_PROGRAM
```

#### Revision.var - Local variables
```iecst
(********************************************************************
 * COPYRIGHT --
 ********************************************************************
 * Program: Revision
 * File: Revision.var
 * Author: pkiel
 * Created: December 14, 2009
 ********************************************************************
 * Local variables of program Revision
 ********************************************************************)
VAR
	CurrentSoftwareRevision : REAL;
END_VAR
```

### Program Logical/SupervisoryControl_Section/Run
